LIN {X 0,Y 418.595,Z 415.277,A -85,B 0,C 180,E1 -16911.483,E2 -16911.483} C_VEL
LIN {X 0,Y 414.654,Z 412.078,A -85,B 0,C 180,E1 -16916.405,E2 -16916.405} C_VEL
LIN {X 0,Y 413.753,Z 409.569,A -85,B 0,C 180,E1 -16920.138,E2 -16920.138} C_VEL
LIN {X 0,Y 413.822,Z 409.954,A -85,B 0,C 180,E1 -16922.354,E2 -16922.354} C_VEL
LIN {X 0,Y 418.138,Z 415.092,A -85,B 0,C 180,E1 -16929.775,E2 -16929.775} C_VEL
LIN {X 0,Y 418.882,Z 415.623,A -85,B 0,C 180,E1 -16930.452,E2 -16930.452} C_VEL
LIN {X 0,Y 421.003,Z 419.369,A -85,B 0,C 180,E1 -16932.342,E2 -16932.342} C_VEL
LIN {X 0,Y 424.072,Z 421.923,A -85,B 0,C 180,E1 -16934.404,E2 -16934.404} C_VEL
LIN {X 0,Y 426.834,Z 426.008,A -85,B 0,C 180,E1 -16936.117,E2 -16936.117} C_VEL
LIN {X 0,Y 429.181,Z 428.229,A -85,B 0,C 180,E1 -16937.35,E2 -16937.35} C_VEL
LIN {X 0,Y 432.702,Z 432.705,A -85,B 0,C 180,E1 -16939.086,E2 -16939.086} C_VEL
LIN {X 0,Y 434.181,Z 434.42,A -85,B 0,C 180,E1 -16939.752,E2 -16939.752} C_VEL
LIN {X 0,Y 438.948,Z 440.495,A -85,B 0,C 180,E1 -16941.761,E2 -16941.761} C_VEL
LIN {X 0,Y 444.689,Z 448.712,A -85,B 0,C 180,E1 -16943.945,E2 -16943.945} C_VEL
LIN {X 0,Y 452.263,Z 459.705,A -85,B 0,C 180,E1 -16946.49,E2 -16946.49} C_VEL
LIN {X 0,Y 462.215,Z 475.454,A -85,B 0,C 180,E1 -16949.446,E2 -16949.446} C_VEL
LIN {X 0,Y 471.304,Z 490.869,A -85,B 0,C 180,E1 -16951.853,E2 -16951.853} C_VEL
LIN {X 0,Y 477.792,Z 502.788,A -85,B 0,C 180,E1 -16953.445,E2 -16953.445} C_VEL
LIN {X 0,Y 463.026,Z 751.514,A -85,B 0,C 180,E1 -16957.403,E2 -16957.403} C_VEL
LIN {X 0,Y 460.977,Z 774.068,A -85,B 0,C 180,E1 -16957.838,E2 -16957.838} C_VEL
LIN {X 0,Y 457.627,Z 798.83,A -85,B 0,C 180,E1 -16958.465,E2 -16958.465} C_VEL
LIN {X 0,Y 453.795,Z 820.475,A -85,B 0,C 180,E1 -16959.196,E2 -16959.196} C_VEL
LIN {X 0,Y 449.461,Z 841.373,A -85,B 0,C 180,E1 -16960.068,E2 -16960.068} C_VEL
LIN {X 0,Y 443.769,Z 864.79,A -85,B 0,C 180,E1 -16961.285,E2 -16961.285} C_VEL
LIN {X 0,Y 438.553,Z 883.81,A -85,B 0,C 180,E1 -16962.475,E2 -16962.475} C_VEL
LIN {X 0,Y 431.836,Z 906.004,A -85,B 0,C 180,E1 -16964.128,E2 -16964.128} C_VEL
LIN {X 0,Y 425.724,Z 924.421,A -85,B 0,C 180,E1 -16965.769,E2 -16965.769} C_VEL
LIN {X 0,Y 418.908,Z 943.868,A -85,B 0,C 180,E1 -16967.785,E2 -16967.785} C_VEL
LIN {X 0,Y 412.181,Z 961.726,A -85,B 0,C 180,E1 -16969.995,E2 -16969.995} C_VEL
LIN {X 0,Y 405.9,Z 978.095,A -85,B 0,C 180,E1 -16972.344,E2 -16972.344} C_VEL
LIN {X 0,Y 399.636,Z 994.038,A -85,B 0,C 180,E1 -16975.043,E2 -16975.043} C_VEL
LIN {X 0,Y 394.447,Z 1007.349,A -85,B 0,C 180,E1 -16977.665,E2 -16977.665} C_VEL
LIN {X 0,Y 388.853,Z 1022.095,A -85,B 0,C 180,E1 -16981.091,E2 -16981.091} C_VEL
LIN {X 0,Y 384.923,Z 1033.094,A -85,B 0,C 180,E1 -16984.125,E2 -16984.125} C_VEL
LIN {X 0,Y 381.161,Z 1044.727,A -85,B 0,C 180,E1 -16987.968,E2 -16987.968} C_VEL
LIN {X 0,Y 378.92,Z 1052.817,A -85,B 0,C 180,E1 -16991.22,E2 -16991.22} C_VEL
LIN {X 0,Y 377.195,Z 1060.626,A -85,B 0,C 180,E1 -16995.1,E2 -16995.1} C_VEL
LIN {X 0,Y 376.396,Z 1065.668,A -85,B 0,C 180,E1 -16998.352,E2 -16998.352} C_VEL
LIN {X 0,Y 376.025,Z 1069.646,A -85,B 0,C 180,E1 -17001.744,E2 -17001.744} C_VEL
LIN {X 0,Y 375.948,Z 1072.336,A -85,B 0,C 180,E1 -17005.424,E2 -17005.424} C_VEL
LIN {X 0,Y 375.957,Z 1073.33,A -85,B 0,C 180,E1 -17008.324,E2 -17008.324} C_VEL
LIN {X 0,Y 375.965,Z 1073.331,A -85,B 0,C 180,E1 -17011.219,E2 -17011.219} C_VEL
LIN {X 0,Y 375.951,Z 1072.197,A -85,B 0,C 180,E1 -17014.424,E2 -17014.424} C_VEL
LIN {X 0,Y 376.015,Z 1069.299,A -85,B 0,C 180,E1 -17018.102,E2 -17018.102} C_VEL
LIN {X 0,Y 376.313,Z 1065.625,A -85,B 0,C 180,E1 -17021.184,E2 -17021.184} C_VEL
LIN {X 0,Y 377.065,Z 1060.282,A -85,B 0,C 180,E1 -17024.591,E2 -17024.591} C_VEL
LIN {X 0,Y 378.591,Z 1052.628,A -85,B 0,C 180,E1 -17028.318,E2 -17028.318} C_VEL
LIN {X 0,Y 380.669,Z 1044.446,A -85,B 0,C 180,E1 -17031.576,E2 -17031.576} C_VEL
LIN {X 0,Y 384.037,Z 1033.144,A -85,B 0,C 180,E1 -17035.277,E2 -17035.277} C_VEL
LIN {X 0,Y 387.534,Z 1022.627,A -85,B 0,C 180,E1 -17038.175,E2 -17038.175} C_VEL
LIN {X 0,Y 392.523,Z 1008.535,A -85,B 0,C 180,E1 -17041.48,E2 -17041.48} C_VEL
LIN {X 0,Y 397.395,Z 995.196,A -85,B 0,C 180,E1 -17044.131,E2 -17044.131} C_VEL
LIN {X 0,Y 403.31,Z 979.283,A -85,B 0,C 180,E1 -17046.868,E2 -17046.868} C_VEL
LIN {X 0,Y 409.632,Z 961.81,A -85,B 0,C 180,E1 -17049.394,E2 -17049.394} C_VEL
LIN {X 0,Y 416.292,Z 943.126,A -85,B 0,C 180,E1 -17051.707,E2 -17051.707} C_VEL
LIN {X 0,Y 422.435,Z 924.703,A -85,B 0,C 180,E1 -17053.628,E2 -17053.628} C_VEL
LIN {X 0,Y 428.561,Z 905.351,A -85,B 0,C 180,E1 -17055.366,E2 -17055.366} C_VEL
LIN {X 0,Y 434.811,Z 883.629,A -85,B 0,C 180,E1 -17056.993,E2 -17056.993} C_VEL
LIN {X 0,Y 439.864,Z 864.356,A -85,B 0,C 180,E1 -17058.211,E2 -17058.211} C_VEL
LIN {X 0,Y 445.381,Z 840.47,A -85,B 0,C 180,E1 -17059.459,E2 -17059.459} C_VEL
LIN {X 0,Y 449.404,Z 820.168,A -85,B 0,C 180,E1 -17060.316,E2 -17060.316} C_VEL
LIN {X 0,Y 453.43,Z 796.266,A -85,B 0,C 180,E1 -17061.123,E2 -17061.123} C_VEL
LIN {X 0,Y 456.393,Z 772.598,A -85,B 0,C 180,E1 -17061.714,E2 -17061.714} C_VEL
LIN {X 0,Y 458.46,Z 747.708,A -85,B 0,C 180,E1 -17062.189,E2 -17062.189} C_VEL
LIN {X 0,Y 472.43,Z 499.373,A -85,B 0,C 180,E1 -17066.15,E2 -17066.15} C_VEL
LIN {X 0,Y 462.964,Z 482.094,A -85,B 0,C 180,E1 -17068.344,E2 -17068.344} C_VEL
LIN {X 0,Y 452.861,Z 465.203,A -85,B 0,C 180,E1 -17070.902,E2 -17070.902} C_VEL
LIN {X 0,Y 442.865,Z 449.591,A -85,B 0,C 180,E1 -17073.735,E2 -17073.735} C_VEL
LIN {X 0,Y 433.988,Z 436.811,A -85,B 0,C 180,E1 -17076.582,E2 -17076.582} C_VEL
LIN {X 0,Y 429.245,Z 430.714,A -85,B 0,C 180,E1 -17078.261,E2 -17078.261} C_VEL
LIN {X 0,Y 424.967,Z 425.414,A -85,B 0,C 180,E1 -17079.908,E2 -17079.908} C_VEL
LIN {X 0,Y 421.299,Z 420.825,A -85,B 0,C 180,E1 -17081.456,E2 -17081.456} C_VEL
LIN {X 0,Y 416.853,Z 415.708,A -85,B 0,C 180,E1 -17083.522,E2 -17083.522} C_VEL
LIN {X 0,Y 415.772,Z 414.109,A -85,B 0,C 180,E1 -17084.088,E2 -17084.088} C_VEL
LIN {X 0,Y 412.366,Z 410.911,A -85,B 0,C 180,E1 -17085.908,E2 -17085.908} C_VEL
LIN {X 0,Y 410.586,Z 407.937,A -85,B 0,C 180,E1 -17087.053,E2 -17087.053} C_VEL
LIN {X 0,Y 407.105,Z 405.166,A -85,B 0,C 180,E1 -17089.385,E2 -17089.385} C_VEL
LIN {X 0,Y 405.262,Z 401.53,A -85,B 0,C 180,E1 -17091.058,E2 -17091.058} C_VEL
LIN {X 0,Y 401.47,Z 399.131,A -85,B 0,C 180,E1 -17095.142,E2 -17095.142} C_VEL
LIN {X 0,Y 399.74,Z 395.247,A -85,B 0,C 180,E1 -17100.43,E2 -17100.43} C_VEL
LIN {X 0,Y 399.742,Z 395.247,A -85,B 0,C 180,E1 -17102.007,E2 -17102.007} C_VEL
LIN {X 0,Y 401.877,Z 399.568,A -85,B 0,C 180,E1 -17107.865,E2 -17107.865} C_VEL
LIN {X 0,Y 405.347,Z 401.809,A -85,B 0,C 180,E1 -17111.454,E2 -17111.454} C_VEL
LIN {X 0,Y 407.325,Z 405.383,A -85,B 0,C 180,E1 -17113.197,E2 -17113.197} C_VEL
LIN {X 0,Y 410.405,Z 407.832,A -85,B 0,C 180,E1 -17115.256,E2 -17115.256} C_VEL
LIN {X 0,Y 411.097,Z 408.742,A -85,B 0,C 180,E1 -17115.699,E2 -17115.699} C_VEL
LIN {X 0,Y 413.993,Z 412.767,A -85,B 0,C 180,E1 -17117.427,E2 -17117.427} C_VEL
LIN {X 0,Y 416.281,Z 414.792,A -85,B 0,C 180,E1 -17118.594,E2 -17118.594} C_VEL
LIN {X 0,Y 419.453,Z 418.976,A -85,B 0,C 180,E1 -17120.149,E2 -17120.149} C_VEL
LIN {X 0,Y 421.308,Z 420.811,A -85,B 0,C 180,E1 -17120.964,E2 -17120.964} C_VEL
LIN {X 0,Y 425.07,Z 425.454,A -85,B 0,C 180,E1 -17122.546,E2 -17122.546} C_VEL
LIN {X 0,Y 427.658,Z 428.844,A -85,B 0,C 180,E1 -17123.566,E2 -17123.566} C_VEL
LIN {X 0,Y 431.094,Z 432.964,A -85,B 0,C 180,E1 -17124.823,E2 -17124.823} C_VEL
LIN {X 0,Y 435.975,Z 439.247,A -85,B 0,C 180,E1 -17126.492,E2 -17126.492} C_VEL
LIN {X 0,Y 442.658,Z 447.991,A -85,B 0,C 180,E1 -17128.575,E2 -17128.575} C_VEL
LIN {X 0,Y 452.49,Z 461.584,A -85,B 0,C 180,E1 -17131.322,E2 -17131.322} C_VEL
LIN {X 0,Y 462.744,Z 476.797,A -85,B 0,C 180,E1 -17133.882,E2 -17133.882} C_VEL
LIN {X 0,Y 472.66,Z 492.479,A -85,B 0,C 180,E1 -17136.128,E2 -17136.128} C_VEL
LIN {X 0,Y 458.588,Z 739.184,A -85,B 0,C 180,E1 -17140.069,E2 -17140.069} C_VEL
LIN {X 0,Y 456.64,Z 761.14,A -85,B 0,C 180,E1 -17140.516,E2 -17140.516} C_VEL
LIN {X 0,Y 453.326,Z 786.702,A -85,B 0,C 180,E1 -17141.231,E2 -17141.231} C_VEL
LIN {X 0,Y 450.006,Z 806.703,A -85,B 0,C 180,E1 -17141.956,E2 -17141.956} C_VEL
LIN {X 0,Y 445.549,Z 829.565,A -85,B 0,C 180,E1 -17142.979,E2 -17142.979} C_VEL
LIN {X 0,Y 440.536,Z 851.049,A -85,B 0,C 180,E1 -17144.174,E2 -17144.174} C_VEL
LIN {X 0,Y 435.215,Z 871.436,A -85,B 0,C 180,E1 -17145.515,E2 -17145.515} C_VEL
LIN {X 0,Y 428.993,Z 892.708,A -85,B 0,C 180,E1 -17147.201,E2 -17147.201} C_VEL
LIN {X 0,Y 423.304,Z 910.614,A -85,B 0,C 180,E1 -17148.864,E2 -17148.864} C_VEL
LIN {X 0,Y 416.422,Z 930.803,A -85,B 0,C 180,E1 -17151.076,E2 -17151.076} C_VEL
LIN {X 0,Y 410.742,Z 946.551,A -85,B 0,C 180,E1 -17153.099,E2 -17153.099} C_VEL
LIN {X 0,Y 404.223,Z 964.023,A -85,B 0,C 180,E1 -17155.709,E2 -17155.709} C_VEL
LIN {X 0,Y 398.77,Z 978.285,A -85,B 0,C 180,E1 -17158.227,E2 -17158.227} C_VEL
LIN {X 0,Y 393.418,Z 992.492,A -85,B 0,C 180,E1 -17161.126,E2 -17161.126} C_VEL
LIN {X 0,Y 388.636,Z 1005.189,A -85,B 0,C 180,E1 -17164.227,E2 -17164.227} C_VEL
LIN {X 0,Y 384.759,Z 1016.241,A -85,B 0,C 180,E1 -17167.38,E2 -17167.38} C_VEL
LIN {X 0,Y 381.461,Z 1026.344,A -85,B 0,C 180,E1 -17170.874,E2 -17170.874} C_VEL
LIN {X 0,Y 379.252,Z 1034.079,A -85,B 0,C 180,E1 -17174.086,E2 -17174.086} C_VEL
LIN {X 0,Y 377.506,Z 1041.462,A -85,B 0,C 180,E1 -17177.922,E2 -17177.922} C_VEL
LIN {X 0,Y 376.635,Z 1046.231,A -85,B 0,C 180,E1 -17181.142,E2 -17181.142} C_VEL
LIN {X 0,Y 376.175,Z 1050.124,A -85,B 0,C 180,E1 -17184.662,E2 -17184.662} C_VEL
LIN {X 0,Y 376.006,Z 1052.412,A -85,B 0,C 180,E1 -17188.171,E2 -17188.171} C_VEL
LIN {X 0,Y 375.97,Z 1053.298,A -85,B 0,C 180,E1 -17191.067,E2 -17191.067} C_VEL
LIN {X 0,Y 375.98,Z 1053.205,A -85,B 0,C 180,E1 -17194.219,E2 -17194.219} C_VEL
LIN {X 0,Y 376.077,Z 1051.718,A -85,B 0,C 180,E1 -17197.793,E2 -17197.793} C_VEL
LIN {X 0,Y 376.362,Z 1049.06,A -85,B 0,C 180,E1 -17201.028,E2 -17201.028} C_VEL
LIN {X 0,Y 376.991,Z 1045.229,A -85,B 0,C 180,E1 -17204.28,E2 -17204.28} C_VEL
LIN {X 0,Y 378.403,Z 1038.971,A -85,B 0,C 180,E1 -17208.168,E2 -17208.168} C_VEL
LIN {X 0,Y 380.312,Z 1032.182,A -85,B 0,C 180,E1 -17211.453,E2 -17211.453} C_VEL
LIN {X 0,Y 383.447,Z 1022.659,A -85,B 0,C 180,E1 -17215.196,E2 -17215.196} C_VEL
LIN {X 0,Y 384.449,Z 1019.742,A -85,B 0,C 180,E1 -17216.188,E2 -17216.188} C_VEL
LIN {X 0,Y 384.646,Z 1016.77,A -85,B 0,C 180,E1 -17217.254,E2 -17217.254} C_VEL
LIN {X 0,Y 382.131,Z 1008.67,A -85,B 0,C 180,E1 -17220.166,E2 -17220.166} C_VEL
LIN {X 0,Y 382.694,Z 1005.603,A -85,B 0,C 180,E1 -17221.052,E2 -17221.052} C_VEL
LIN {X 0,Y 388.256,Z 992.368,A -85,B 0,C 180,E1 -17224.333,E2 -17224.333} C_VEL
LIN {X 0,Y 394.017,Z 978.627,A -85,B 0,C 180,E1 -17227.171,E2 -17227.171} C_VEL
LIN {X 0,Y 400.549,Z 963.213,A -85,B 0,C 180,E1 -17229.907,E2 -17229.907} C_VEL
LIN {X 0,Y 407.452,Z 946.166,A -85,B 0,C 180,E1 -17232.443,E2 -17232.443} C_VEL
LIN {X 0,Y 414.186,Z 929.038,A -85,B 0,C 180,E1 -17234.628,E2 -17234.628} C_VEL
LIN {X 0,Y 421.151,Z 910.027,A -85,B 0,C 180,E1 -17236.674,E2 -17236.674} C_VEL
LIN {X 0,Y 427.212,Z 892.368,A -85,B 0,C 180,E1 -17238.298,E2 -17238.298} C_VEL
LIN {X 0,Y 434.282,Z 869.687,A -85,B 0,C 180,E1 -17240.058,E2 -17240.058} C_VEL
LIN {X 0,Y 439.772,Z 850.01,A -85,B 0,C 180,E1 -17241.325,E2 -17241.325} C_VEL
LIN {X 0,Y 445.565,Z 826.246,A -85,B 0,C 180,E1 -17242.6,E2 -17242.6} C_VEL
LIN {X 0,Y 449.848,Z 805.433,A -85,B 0,C 180,E1 -17243.498,E2 -17243.498} C_VEL
LIN {X 0,Y 453.959,Z 781.735,A -85,B 0,C 180,E1 -17244.321,E2 -17244.321} C_VEL
LIN {X 0,Y 457.039,Z 757.598,A -85,B 0,C 180,E1 -17244.941,E2 -17244.941} C_VEL
LIN {X 0,Y 459.217,Z 732.893,A -85,B 0,C 180,E1 -17245.412,E2 -17245.412} C_VEL
LIN {X 0,Y 473.455,Z 500.104,A -85,B 0,C 180,E1 -17249.123,E2 -17249.123} C_VEL
LIN {X 0,Y 463.328,Z 484.174,A -85,B 0,C 180,E1 -17251.697,E2 -17251.697} C_VEL
LIN {X 0,Y 453.867,Z 470.442,A -85,B 0,C 180,E1 -17254.383,E2 -17254.383} C_VEL
LIN {X 0,Y 446.179,Z 459.921,A -85,B 0,C 180,E1 -17256.84,E2 -17256.84} C_VEL
LIN {X 0,Y 439.936,Z 451.462,A -85,B 0,C 180,E1 -17259.094,E2 -17259.094} C_VEL
LIN {X 0,Y 435.12,Z 445.449,A -85,B 0,C 180,E1 -17261.025,E2 -17261.025} C_VEL
LIN {X 0,Y 431.297,Z 440.548,A -85,B 0,C 180,E1 -17262.738,E2 -17262.738} C_VEL
LIN {X 0,Y 427.805,Z 436.18,A -85,B 0,C 180,E1 -17264.477,E2 -17264.477} C_VEL
LIN {X 0,Y 426.589,Z 434.763,A -85,B 0,C 180,E1 -17265.128,E2 -17265.128} C_VEL
LIN {X 0,Y 423.245,Z 430.774,A -85,B 0,C 180,E1 -17267.1,E2 -17267.1} C_VEL
LIN {X 0,Y 422.373,Z 429.307,A -85,B 0,C 180,E1 -17267.698,E2 -17267.698} C_VEL
LIN {X 0,Y 418.943,Z 426.044,A -85,B 0,C 180,E1 -17270.174,E2 -17270.174} C_VEL
LIN {X 0,Y 417.474,Z 423.172,A -85,B 0,C 180,E1 -17271.599,E2 -17271.599} C_VEL
LIN {X 0,Y 413.613,Z 419.955,A -85,B 0,C 180,E1 -17276.535,E2 -17276.535} C_VEL
LIN {X 0,Y 412.773,Z 417.456,A -85,B 0,C 180,E1 -17280.278,E2 -17280.278} C_VEL
LIN {X 0,Y 412.842,Z 417.936,A -85,B 0,C 180,E1 -17282.36,E2 -17282.36} C_VEL
LIN {X 0,Y 417.027,Z 422.988,A -85,B 0,C 180,E1 -17289.662,E2 -17289.662} C_VEL
LIN {X 0,Y 417.682,Z 423.496,A -85,B 0,C 180,E1 -17290.273,E2 -17290.273} C_VEL
LIN {X 0,Y 419.856,Z 427.269,A -85,B 0,C 180,E1 -17292.237,E2 -17292.237} C_VEL
LIN {X 0,Y 422.682,Z 429.677,A -85,B 0,C 180,E1 -17294.172,E2 -17294.172} C_VEL
LIN {X 0,Y 425.518,Z 433.819,A -85,B 0,C 180,E1 -17295.958,E2 -17295.958} C_VEL
LIN {X 0,Y 427.645,Z 435.902,A -85,B 0,C 180,E1 -17297.099,E2 -17297.099} C_VEL
LIN {X 0,Y 431.324,Z 440.528,A -85,B 0,C 180,E1 -17298.938,E2 -17298.938} C_VEL
LIN {X 0,Y 437.04,Z 447.87,A -85,B 0,C 180,E1 -17301.438,E2 -17301.438} C_VEL
LIN {X 0,Y 442.601,Z 455.989,A -85,B 0,C 180,E1 -17303.605,E2 -17303.605} C_VEL
LIN {X 0,Y 449.951,Z 466.899,A -85,B 0,C 180,E1 -17306.136,E2 -17306.136} C_VEL
LIN {X 0,Y 459.467,Z 482.19,A -85,B 0,C 180,E1 -17309.032,E2 -17309.032} C_VEL
LIN {X 0,Y 468.305,Z 497.46,A -85,B 0,C 180,E1 -17311.433,E2 -17311.433} C_VEL
LIN {X 0,Y 473.26,Z 506.669,A -85,B 0,C 180,E1 -17312.69,E2 -17312.69} C_VEL
LIN {X 0,Y 458.137,Z 753.356,A -85,B 0,C 180,E1 -17316.632,E2 -17316.632} C_VEL
LIN {X 0,Y 455.983,Z 775.737,A -85,B 0,C 180,E1 -17317.072,E2 -17317.072} C_VEL
LIN {X 0,Y 452.153,Z 802.073,A -85,B 0,C 180,E1 -17317.764,E2 -17317.764} C_VEL
LIN {X 0,Y 448.34,Z 822.781,A -85,B 0,C 180,E1 -17318.482,E2 -17318.482} C_VEL
LIN {X 0,Y 443.19,Z 846.317,A -85,B 0,C 180,E1 -17319.503,E2 -17319.503} C_VEL
LIN {X 0,Y 437.935,Z 866.84,A -85,B 0,C 180,E1 -17320.61,E2 -17320.61} C_VEL
LIN {X 0,Y 432.081,Z 887.426,A -85,B 0,C 180,E1 -17321.928,E2 -17321.928} C_VEL
LIN {X 0,Y 425.546,Z 907.928,A -85,B 0,C 180,E1 -17323.508,E2 -17323.508} C_VEL
LIN {X 0,Y 419.209,Z 926.381,A -85,B 0,C 180,E1 -17325.185,E2 -17325.185} C_VEL
LIN {X 0,Y 411.637,Z 946.918,A -85,B 0,C 180,E1 -17327.393,E2 -17327.393} C_VEL
LIN {X 0,Y 405.349,Z 963.072,A -85,B 0,C 180,E1 -17329.443,E2 -17329.443} C_VEL
LIN {X 0,Y 398.317,Z 980.667,A -85,B 0,C 180,E1 -17332.047,E2 -17332.047} C_VEL
LIN {X 0,Y 392.19,Z 995.609,A -85,B 0,C 180,E1 -17334.671,E2 -17334.671} C_VEL
LIN {X 0,Y 386.377,Z 1010.038,A -85,B 0,C 180,E1 -17337.609,E2 -17337.609} C_VEL
LIN {X 0,Y 381.166,Z 1023.104,A -85,B 0,C 180,E1 -17340.796,E2 -17340.796} C_VEL
LIN {X 0,Y 376.92,Z 1034.573,A -85,B 0,C 180,E1 -17344.066,E2 -17344.066} C_VEL
LIN {X 0,Y 373.388,Z 1044.968,A -85,B 0,C 180,E1 -17347.65,E2 -17347.65} C_VEL
LIN {X 0,Y 371.048,Z 1053,A -85,B 0,C 180,E1 -17350.97,E2 -17350.97} C_VEL
LIN {X 0,Y 369.244,Z 1060.698,A -85,B 0,C 180,E1 -17354.932,E2 -17354.932} C_VEL
LIN {X 0,Y 368.41,Z 1065.687,A -85,B 0,C 180,E1 -17358.255,E2 -17358.255} C_VEL
LIN {X 0,Y 368.013,Z 1069.776,A -85,B 0,C 180,E1 -17361.878,E2 -17361.878} C_VEL
LIN {X 0,Y 367.949,Z 1072.2,A -85,B 0,C 180,E1 -17365.48,E2 -17365.48} C_VEL
LIN {X 0,Y 367.96,Z 1073.142,A -85,B 0,C 180,E1 -17368.443,E2 -17368.443} C_VEL
LIN {X 0,Y 367.964,Z 1073.092,A -85,B 0,C 180,E1 -17371.401,E2 -17371.401} C_VEL
LIN {X 0,Y 367.957,Z 1071.742,A -85,B 0,C 180,E1 -17374.989,E2 -17374.989} C_VEL
LIN {X 0,Y 368.049,Z 1068.787,A -85,B 0,C 180,E1 -17378.546,E2 -17378.546} C_VEL
LIN {X 0,Y 368.399,Z 1064.96,A -85,B 0,C 180,E1 -17381.745,E2 -17381.745} C_VEL
LIN {X 0,Y 369.37,Z 1058.884,A -85,B 0,C 180,E1 -17385.545,E2 -17385.545} C_VEL
LIN {X 0,Y 370.963,Z 1051.643,A -85,B 0,C 180,E1 -17389.035,E2 -17389.035} C_VEL
LIN {X 0,Y 373.52,Z 1042.506,A -85,B 0,C 180,E1 -17392.673,E2 -17392.673} C_VEL
LIN {X 0,Y 376.915,Z 1031.81,A -85,B 0,C 180,E1 -17396.127,E2 -17396.127} C_VEL
LIN {X 0,Y 381.193,Z 1019.77,A -85,B 0,C 180,E1 -17399.441,E2 -17399.441} C_VEL
LIN {X 0,Y 386.259,Z 1006.087,A -85,B 0,C 180,E1 -17402.577,E2 -17402.577} C_VEL
LIN {X 0,Y 391.772,Z 991.744,A -85,B 0,C 180,E1 -17405.405,E2 -17405.405} C_VEL
LIN {X 0,Y 398.151,Z 975.046,A -85,B 0,C 180,E1 -17408.182,E2 -17408.182} C_VEL
LIN {X 0,Y 404.06,Z 959.404,A -85,B 0,C 180,E1 -17410.417,E2 -17410.417} C_VEL
LIN {X 0,Y 411.225,Z 939.668,A -85,B 0,C 180,E1 -17412.812,E2 -17412.812} C_VEL
LIN {X 0,Y 417.284,Z 922.041,A -85,B 0,C 180,E1 -17414.629,E2 -17414.629} C_VEL
LIN {X 0,Y 424.273,Z 900.17,A -85,B 0,C 180,E1 -17416.541,E2 -17416.541} C_VEL
LIN {X 0,Y 429.916,Z 880.895,A -85,B 0,C 180,E1 -17417.946,E2 -17417.946} C_VEL
LIN {X 0,Y 435.801,Z 858.702,A -85,B 0,C 180,E1 -17419.314,E2 -17419.314} C_VEL
LIN {X 0,Y 440.76,Z 836.985,A -85,B 0,C 180,E1 -17420.397,E2 -17420.397} C_VEL
LIN {X 0,Y 444.916,Z 816.254,A -85,B 0,C 180,E1 -17421.245,E2 -17421.245} C_VEL
LIN {X 0,Y 449.001,Z 791.127,A -85,B 0,C 180,E1 -17422.045,E2 -17422.045} C_VEL
LIN {X 0,Y 451.686,Z 769.398,A -85,B 0,C 180,E1 -17422.569,E2 -17422.569} C_VEL
LIN {X 0,Y 454.074,Z 736.841,A -85,B 0,C 180,E1 -17423.153,E2 -17423.153} C_VEL
LIN {X 0,Y 467.644,Z 503.033,A -85,B 0,C 180,E1 -17426.899,E2 -17426.899} C_VEL
LIN {X 0,Y 457.829,Z 485.159,A -85,B 0,C 180,E1 -17429.266,E2 -17429.266} C_VEL
LIN {X 0,Y 448.434,Z 469.378,A -85,B 0,C 180,E1 -17431.754,E2 -17431.754} C_VEL
LIN {X 0,Y 439.686,Z 455.676,A -85,B 0,C 180,E1 -17434.328,E2 -17434.328} C_VEL
LIN {X 0,Y 431.475,Z 443.557,A -85,B 0,C 180,E1 -17437.052,E2 -17437.052} C_VEL
LIN {X 0,Y 427.074,Z 437.891,A -85,B 0,C 180,E1 -17438.65,E2 -17438.65} C_VEL
LIN {X 0,Y 423.034,Z 432.801,A -85,B 0,C 180,E1 -17440.245,E2 -17440.245} C_VEL
LIN {X 0,Y 419.299,Z 427.956,A -85,B 0,C 180,E1 -17441.868,E2 -17441.868} C_VEL
LIN {X 0,Y 415.399,Z 423.561,A -85,B 0,C 180,E1 -17443.715,E2 -17443.715} C_VEL
LIN {X 0,Y 414.009,Z 421.639,A -85,B 0,C 180,E1 -17444.45,E2 -17444.45} C_VEL
LIN {X 0,Y 410.724,Z 418.316,A -85,B 0,C 180,E1 -17446.269,E2 -17446.269} C_VEL
LIN {X 0,Y 409.172,Z 415.703,A -85,B 0,C 180,E1 -17447.295,E2 -17447.295} C_VEL
LIN {X 0,Y 405.686,Z 412.733,A -85,B 0,C 180,E1 -17449.707,E2 -17449.707} C_VEL
LIN {X 0,Y 403.962,Z 409.372,A -85,B 0,C 180,E1 -17451.316,E2 -17451.316} C_VEL
LIN {X 0,Y 400.228,Z 406.777,A -85,B 0,C 180,E1 -17455.558,E2 -17455.558} C_VEL
LIN {X 0,Y 398.765,Z 403.19,A -85,B 0,C 180,E1 -17460.431,E2 -17460.431} C_VEL
LIN {X 0,Y 398.764,Z 403.218,A -85,B 0,C 180,E1 -17462.012,E2 -17462.012} C_VEL
LIN {X 0,Y 402.905,Z 408.947,A -85,B 0,C 180,E1 -17470.149,E2 -17470.149} C_VEL
LIN {X 0,Y 404.064,Z 409.552,A -85,B 0,C 180,E1 -17471.201,E2 -17471.201} C_VEL
LIN {X 0,Y 406.171,Z 413.304,A -85,B 0,C 180,E1 -17473.09,E2 -17473.09} C_VEL
LIN {X 0,Y 409.485,Z 416.11,A -85,B 0,C 180,E1 -17475.327,E2 -17475.327} C_VEL
LIN {X 0,Y 412.414,Z 420.34,A -85,B 0,C 180,E1 -17477.132,E2 -17477.132} C_VEL
LIN {X 0,Y 414.717,Z 422.496,A -85,B 0,C 180,E1 -17478.339,E2 -17478.339} C_VEL
LIN {X 0,Y 418.065,Z 426.807,A -85,B 0,C 180,E1 -17480,E2 -17480} C_VEL
LIN {X 0,Y 419.667,Z 428.537,A -85,B 0,C 180,E1 -17480.721,E2 -17480.721} C_VEL
LIN {X 0,Y 423.636,Z 433.301,A -85,B 0,C 180,E1 -17482.407,E2 -17482.407} C_VEL
LIN {X 0,Y 429.418,Z 440.849,A -85,B 0,C 180,E1 -17484.633,E2 -17484.633} C_VEL
LIN {X 0,Y 434.165,Z 447.01,A -85,B 0,C 180,E1 -17486.28,E2 -17486.28} C_VEL
LIN {X 0,Y 440.974,Z 456.175,A -85,B 0,C 180,E1 -17488.436,E2 -17488.436} C_VEL
LIN {X 0,Y 449.772,Z 468.497,A -85,B 0,C 180,E1 -17490.937,E2 -17490.937} C_VEL
LIN {X 0,Y 459.776,Z 483.553,A -85,B 0,C 180,E1 -17493.493,E2 -17493.493} C_VEL
LIN {X 0,Y 467.865,Z 496.717,A -85,B 0,C 180,E1 -17495.389,E2 -17495.389} C_VEL
LIN {X 0,Y 453.549,Z 740.077,A -85,B 0,C 180,E1 -17499.294,E2 -17499.294} C_VEL
LIN {X 0,Y 451.468,Z 762.645,A -85,B 0,C 180,E1 -17499.76,E2 -17499.76} C_VEL
LIN {X 0,Y 448.099,Z 787.565,A -85,B 0,C 180,E1 -17500.469,E2 -17500.469} C_VEL
LIN {X 0,Y 444.73,Z 807.283,A -85,B 0,C 180,E1 -17501.188,E2 -17501.188} C_VEL
LIN {X 0,Y 439.958,Z 830.893,A -85,B 0,C 180,E1 -17502.258,E2 -17502.258} C_VEL
LIN {X 0,Y 434.991,Z 851.578,A -85,B 0,C 180,E1 -17503.417,E2 -17503.417} C_VEL
LIN {X 0,Y 429.294,Z 872.789,A -85,B 0,C 180,E1 -17504.824,E2 -17504.824} C_VEL
LIN {X 0,Y 423.117,Z 893.156,A -85,B 0,C 180,E1 -17506.46,E2 -17506.46} C_VEL
LIN {X 0,Y 417.04,Z 911.701,A -85,B 0,C 180,E1 -17508.2,E2 -17508.2} C_VEL
LIN {X 0,Y 410.018,Z 931.561,A -85,B 0,C 180,E1 -17510.409,E2 -17510.409} C_VEL
LIN {X 0,Y 404.138,Z 947.318,A -85,B 0,C 180,E1 -17512.462,E2 -17512.462} C_VEL
LIN {X 0,Y 397.273,Z 965.01,A -85,B 0,C 180,E1 -17515.157,E2 -17515.157} C_VEL
LIN {X 0,Y 391.57,Z 979.385,A -85,B 0,C 180,E1 -17517.745,E2 -17517.745} C_VEL
LIN {X 0,Y 385.699,Z 994.267,A -85,B 0,C 180,E1 -17520.885,E2 -17520.885} C_VEL
LIN {X 0,Y 381.095,Z 1006.064,A -85,B 0,C 180,E1 -17523.846,E2 -17523.846} C_VEL
LIN {X 0,Y 376.909,Z 1017.523,A -85,B 0,C 180,E1 -17527.212,E2 -17527.212} C_VEL
LIN {X 0,Y 373.528,Z 1027.42,A -85,B 0,C 180,E1 -17530.776,E2 -17530.776} C_VEL
LIN {X 0,Y 371.105,Z 1035.73,A -85,B 0,C 180,E1 -17534.369,E2 -17534.369} C_VEL
LIN {X 0,Y 369.496,Z 1042.216,A -85,B 0,C 180,E1 -17537.973,E2 -17537.973} C_VEL
LIN {X 0,Y 368.621,Z 1046.883,A -85,B 0,C 180,E1 -17541.263,E2 -17541.263} C_VEL
LIN {X 0,Y 368.137,Z 1050.811,A -85,B 0,C 180,E1 -17545.17,E2 -17545.17} C_VEL
LIN {X 0,Y 368.003,Z 1052.77,A -85,B 0,C 180,E1 -17548.443,E2 -17548.443} C_VEL
LIN {X 0,Y 367.963,Z 1053.583,A -85,B 0,C 180,E1 -17551.557,E2 -17551.557} C_VEL
LIN {X 0,Y 367.998,Z 1053.234,A -85,B 0,C 180,E1 -17555.144,E2 -17555.144} C_VEL
LIN {X 0,Y 368.14,Z 1051.47,A -85,B 0,C 180,E1 -17558.591,E2 -17558.591} C_VEL
LIN {X 0,Y 368.47,Z 1048.781,A -85,B 0,C 180,E1 -17561.743,E2 -17561.743} C_VEL
LIN {X 0,Y 369.381,Z 1044.115,A -85,B 0,C 180,E1 -17565.545,E2 -17565.545} C_VEL
LIN {X 0,Y 370.849,Z 1038.244,A -85,B 0,C 180,E1 -17569.041,E2 -17569.041} C_VEL
LIN {X 0,Y 373.227,Z 1030.64,A -85,B 0,C 180,E1 -17572.692,E2 -17572.692} C_VEL
LIN {X 0,Y 376.569,Z 1021.105,A -85,B 0,C 180,E1 -17576.323,E2 -17576.323} C_VEL
LIN {X 0,Y 380.596,Z 1010.851,A -85,B 0,C 180,E1 -17579.598,E2 -17579.598} C_VEL
LIN {X 0,Y 382.694,Z 1005.603,A -85,B 0,C 180,E1 -17581.052,E2 -17581.052} C_VEL
LIN {X 0,Y 383.317,Z 1002.103,A -85,B 0,C 180,E1 -17582.081,E2 -17582.081} C_VEL
LIN {X 0,Y 381.972,Z 992.669,A -85,B 0,C 180,E1 -17584.925,E2 -17584.925} C_VEL
LIN {X 0,Y 382.854,Z 989.136,A -85,B 0,C 180,E1 -17585.766,E2 -17585.766} C_VEL
LIN {X 0,Y 388.792,Z 975.723,A -85,B 0,C 180,E1 -17588.49,E2 -17588.49} C_VEL
LIN {X 0,Y 395.749,Z 959.633,A -85,B 0,C 180,E1 -17591.257,E2 -17591.257} C_VEL
LIN {X 0,Y 402.235,Z 944.199,A -85,B 0,C 180,E1 -17593.518,E2 -17593.518} C_VEL
LIN {X 0,Y 409.965,Z 924.952,A -85,B 0,C 180,E1 -17595.912,E2 -17595.912} C_VEL
LIN {X 0,Y 416.614,Z 907.166,A -85,B 0,C 180,E1 -17597.777,E2 -17597.777} C_VEL
LIN {X 0,Y 423.872,Z 886.302,A -85,B 0,C 180,E1 -17599.635,E2 -17599.635} C_VEL
LIN {X 0,Y 429.927,Z 866.82,A -85,B 0,C 180,E1 -17601.084,E2 -17601.084} C_VEL
LIN {X 0,Y 436.219,Z 844.593,A -85,B 0,C 180,E1 -17602.475,E2 -17602.475} C_VEL
LIN {X 0,Y 441.487,Z 822.45,A -85,B 0,C 180,E1 -17603.602,E2 -17603.602} C_VEL
LIN {X 0,Y 445.876,Z 801.155,A -85,B 0,C 180,E1 -17604.492,E2 -17604.492} C_VEL
LIN {X 0,Y 449.985,Z 776.229,A -85,B 0,C 180,E1 -17605.301,E2 -17605.301} C_VEL
LIN {X 0,Y 452.78,Z 754.059,A -85,B 0,C 180,E1 -17605.843,E2 -17605.843} C_VEL
LIN {X 0,Y 455.317,Z 721.258,A -85,B 0,C 180,E1 -17606.422,E2 -17606.422} C_VEL
LIN {X 0,Y 469.023,Z 504.436,A -85,B 0,C 180,E1 -17609.881,E2 -17609.881} C_VEL
LIN {X 0,Y 459.73,Z 489.717,A -85,B 0,C 180,E1 -17612.332,E2 -17612.332} C_VEL
LIN {X 0,Y 451.14,Z 477.063,A -85,B 0,C 180,E1 -17614.85,E2 -17614.85} C_VEL
LIN {X 0,Y 443.696,Z 466.703,A -85,B 0,C 180,E1 -17617.299,E2 -17617.299} C_VEL
LIN {X 0,Y 437.661,Z 458.472,A -85,B 0,C 180,E1 -17619.54,E2 -17619.54} C_VEL
LIN {X 0,Y 433.252,Z 452.826,A -85,B 0,C 180,E1 -17621.359,E2 -17621.359} C_VEL
LIN {X 0,Y 429.5,Z 447.972,A -85,B 0,C 180,E1 -17623.082,E2 -17623.082} C_VEL
LIN {X 0,Y 425.925,Z 443.233,A -85,B 0,C 180,E1 -17624.93,E2 -17624.93} C_VEL
LIN {X 0,Y 421.947,Z 438.647,A -85,B 0,C 180,E1 -17627.268,E2 -17627.268} C_VEL
LIN {X 0,Y 420.99,Z 437.062,A -85,B 0,C 180,E1 -17627.936,E2 -17627.936} C_VEL
LIN {X 0,Y 417.57,Z 433.613,A -85,B 0,C 180,E1 -17630.49,E2 -17630.49} C_VEL
LIN {X 0,Y 416.205,Z 431.007,A -85,B 0,C 180,E1 -17631.851,E2 -17631.851} C_VEL
LIN {X 0,Y 412.17,Z 427.007,A -85,B 0,C 180,E1 -17637.775,E2 -17637.775} C_VEL
LIN {X 0,Y 411.795,Z 425.299,A -85,B 0,C 180,E1 -17640.556,E2 -17640.556} C_VEL
LIN {X 0,Y 411.898,Z 426.108,A -85,B 0,C 180,E1 -17642.644,E2 -17642.644} C_VEL
LIN {X 0,Y 415.919,Z 430.884,A -85,B 0,C 180,E1 -17649.548,E2 -17649.548} C_VEL
LIN {X 0,Y 416.55,Z 431.513,A -85,B 0,C 180,E1 -17650.162,E2 -17650.162} C_VEL
LIN {X 0,Y 418.885,Z 435.355,A -85,B 0,C 180,E1 -17652.266,E2 -17652.266} C_VEL
LIN {X 0,Y 421.301,Z 437.421,A -85,B 0,C 180,E1 -17653.939,E2 -17653.939} C_VEL
LIN {X 0,Y 424.321,Z 441.746,A -85,B 0,C 180,E1 -17655.864,E2 -17655.864} C_VEL
LIN {X 0,Y 426.118,Z 443.564,A -85,B 0,C 180,E1 -17656.846,E2 -17656.846} C_VEL
LIN {X 0,Y 429.95,Z 448.349,A -85,B 0,C 180,E1 -17658.79,E2 -17658.79} C_VEL
LIN {X 0,Y 435.295,Z 455.466,A -85,B 0,C 180,E1 -17661.175,E2 -17661.175} C_VEL
LIN {X 0,Y 440.693,Z 463.515,A -85,B 0,C 180,E1 -17663.324,E2 -17663.324} C_VEL
LIN {X 0,Y 447.764,Z 474.27,A -85,B 0,C 180,E1 -17665.814,E2 -17665.814} C_VEL
LIN {X 0,Y 456.781,Z 488.986,A -85,B 0,C 180,E1 -17668.624,E2 -17668.624} C_VEL
LIN {X 0,Y 465.329,Z 504.068,A -85,B 0,C 180,E1 -17671.009,E2 -17671.009} C_VEL
LIN {X 0,Y 468.796,Z 510.797,A -85,B 0,C 180,E1 -17671.923,E2 -17671.923} C_VEL
LIN {X 0,Y 453.357,Z 754.88,A -85,B 0,C 180,E1 -17675.839,E2 -17675.839} C_VEL
LIN {X 0,Y 450.926,Z 778.675,A -85,B 0,C 180,E1 -17676.316,E2 -17676.316} C_VEL
LIN {X 0,Y 447.1,Z 803.382,A -85,B 0,C 180,E1 -17676.986,E2 -17676.986} C_VEL
LIN {X 0,Y 443.092,Z 824.425,A -85,B 0,C 180,E1 -17677.726,E2 -17677.726} C_VEL
LIN {X 0,Y 437.526,Z 848.652,A -85,B 0,C 180,E1 -17678.804,E2 -17678.804} C_VEL
LIN {X 0,Y 432.44,Z 867.888,A -85,B 0,C 180,E1 -17679.857,E2 -17679.857} C_VEL
LIN {X 0,Y 425.904,Z 890.012,A -85,B 0,C 180,E1 -17681.3,E2 -17681.3} C_VEL
LIN {X 0,Y 419.385,Z 909.625,A -85,B 0,C 180,E1 -17682.85,E2 -17682.85} C_VEL
LIN {X 0,Y 412.739,Z 928.342,A -85,B 0,C 180,E1 -17684.583,E2 -17684.583} C_VEL
LIN {X 0,Y 405.103,Z 948.175,A -85,B 0,C 180,E1 -17686.769,E2 -17686.769} C_VEL
LIN {X 0,Y 398.482,Z 964.6,A -85,B 0,C 180,E1 -17688.896,E2 -17688.896} C_VEL
LIN {X 0,Y 391.099,Z 982.254,A -85,B 0,C 180,E1 -17691.592,E2 -17691.592} C_VEL
LIN {X 0,Y 385.189,Z 996.151,A -85,B 0,C 180,E1 -17694.087,E2 -17694.087} C_VEL
LIN {X 0,Y 378.842,Z 1011.201,A -85,B 0,C 180,E1 -17697.244,E2 -17697.244} C_VEL
LIN {X 0,Y 373.719,Z 1023.535,A -85,B 0,C 180,E1 -17700.332,E2 -17700.332} C_VEL
LIN {X 0,Y 369.151,Z 1035.366,A -85,B 0,C 180,E1 -17703.8,E2 -17703.8} C_VEL
LIN {X 0,Y 365.626,Z 1045.209,A -85,B 0,C 180,E1 -17707.319,E2 -17707.319} C_VEL
LIN {X 0,Y 363.088,Z 1053.541,A -85,B 0,C 180,E1 -17710.87,E2 -17710.87} C_VEL
LIN {X 0,Y 361.296,Z 1060.77,A -85,B 0,C 180,E1 -17714.757,E2 -17714.757} C_VEL
LIN {X 0,Y 360.425,Z 1065.706,A -85,B 0,C 180,E1 -17718.153,E2 -17718.153} C_VEL
LIN {X 0,Y 360.004,Z 1069.826,A -85,B 0,C 180,E1 -17722.017,E2 -17722.017} C_VEL
LIN {X 0,Y 359.952,Z 1071.994,A -85,B 0,C 180,E1 -17725.379,E2 -17725.379} C_VEL
LIN {X 0,Y 359.962,Z 1072.932,A -85,B 0,C 180,E1 -17728.408,E2 -17728.408} C_VEL
LIN {X 0,Y 359.966,Z 1072.875,A -85,B 0,C 180,E1 -17731.432,E2 -17731.432} C_VEL
LIN {X 0,Y 359.958,Z 1071.612,A -85,B 0,C 180,E1 -17734.94,E2 -17734.94} C_VEL
LIN {X 0,Y 360.053,Z 1068.647,A -85,B 0,C 180,E1 -17738.644,E2 -17738.644} C_VEL
LIN {X 0,Y 360.413,Z 1064.93,A -85,B 0,C 180,E1 -17741.847,E2 -17741.847} C_VEL
LIN {X 0,Y 361.408,Z 1059.041,A -85,B 0,C 180,E1 -17745.677,E2 -17745.677} C_VEL
LIN {X 0,Y 363.091,Z 1051.74,A -85,B 0,C 180,E1 -17749.297,E2 -17749.297} C_VEL
LIN {X 0,Y 365.622,Z 1043.077,A -85,B 0,C 180,E1 -17752.851,E2 -17752.851} C_VEL
LIN {X 0,Y 369.3,Z 1032.048,A -85,B 0,C 180,E1 -17756.535,E2 -17756.535} C_VEL
LIN {X 0,Y 373.422,Z 1020.87,A -85,B 0,C 180,E1 -17759.694,E2 -17759.694} C_VEL
LIN {X 0,Y 379.003,Z 1006.487,A -85,B 0,C 180,E1 -17763.1,E2 -17763.1} C_VEL
LIN {X 0,Y 384.385,Z 992.988,A -85,B 0,C 180,E1 -17765.823,E2 -17765.823} C_VEL
LIN {X 0,Y 391.357,Z 975.51,A -85,B 0,C 180,E1 -17768.807,E2 -17768.807} C_VEL
LIN {X 0,Y 397.396,Z 960.08,A -85,B 0,C 180,E1 -17771.049,E2 -17771.049} C_VEL
LIN {X 0,Y 404.992,Z 939.906,A -85,B 0,C 180,E1 -17773.537,E2 -17773.537} C_VEL
LIN {X 0,Y 411.158,Z 922.544,A -85,B 0,C 180,E1 -17775.346,E2 -17775.346} C_VEL
LIN {X 0,Y 418.181,Z 901.381,A -85,B 0,C 180,E1 -17777.227,E2 -17777.227} C_VEL
LIN {X 0,Y 424.222,Z 881.357,A -85,B 0,C 180,E1 -17778.703,E2 -17778.703} C_VEL
LIN {X 0,Y 430.263,Z 859.322,A -85,B 0,C 180,E1 -17780.075,E2 -17780.075} C_VEL
LIN {X 0,Y 435.549,Z 836.78,A -85,B 0,C 180,E1 -17781.205,E2 -17781.205} C_VEL
LIN {X 0,Y 439.892,Z 815.654,A -85,B 0,C 180,E1 -17782.068,E2 -17782.068} C_VEL
LIN {X 0,Y 444.032,Z 790.684,A -85,B 0,C 180,E1 -17782.859,E2 -17782.859} C_VEL
LIN {X 0,Y 446.787,Z 768.832,A -85,B 0,C 180,E1 -17783.384,E2 -17783.384} C_VEL
LIN {X 0,Y 449.223,Z 736.198,A -85,B 0,C 180,E1 -17783.969,E2 -17783.969} C_VEL
LIN {X 0,Y 462.934,Z 506.831,A -85,B 0,C 180,E1 -17787.661,E2 -17787.661} C_VEL
LIN {X 0,Y 453.675,Z 489.843,A -85,B 0,C 180,E1 -17789.98,E2 -17789.98} C_VEL
LIN {X 0,Y 445.019,Z 475.093,A -85,B 0,C 180,E1 -17792.356,E2 -17792.356} C_VEL
LIN {X 0,Y 436.749,Z 462.007,A -85,B 0,C 180,E1 -17794.869,E2 -17794.869} C_VEL
LIN {X 0,Y 429.076,Z 450.432,A -85,B 0,C 180,E1 -17797.495,E2 -17797.495} C_VEL
LIN {X 0,Y 424.757,Z 444.874,A -85,B 0,C 180,E1 -17799.106,E2 -17799.106} C_VEL
LIN {X 0,Y 421.117,Z 440.183,A -85,B 0,C 180,E1 -17800.585,E2 -17800.585} C_VEL
LIN {X 0,Y 416.87,Z 434.813,A -85,B 0,C 180,E1 -17802.481,E2 -17802.481} C_VEL
LIN {X 0,Y 413.273,Z 430.311,A -85,B 0,C 180,E1 -17804.277,E2 -17804.277} C_VEL
LIN {X 0,Y 412.265,Z 429.153,A -85,B 0,C 180,E1 -17804.815,E2 -17804.815} C_VEL
LIN {X 0,Y 408.976,Z 425.523,A -85,B 0,C 180,E1 -17806.714,E2 -17806.714} C_VEL
LIN {X 0,Y 407.766,Z 423.461,A -85,B 0,C 180,E1 -17807.538,E2 -17807.538} C_VEL
LIN {X 0,Y 404.364,Z 420.418,A -85,B 0,C 180,E1 -17809.96,E2 -17809.96} C_VEL
LIN {X 0,Y 402.672,Z 417.207,A -85,B 0,C 180,E1 -17811.576,E2 -17811.576} C_VEL
LIN {X 0,Y 399.086,Z 414.532,A -85,B 0,C 180,E1 -17815.833,E2 -17815.833} C_VEL
LIN {X 0,Y 397.781,Z 411.103,A -85,B 0,C 180,E1 -17820.576,E2 -17820.576} C_VEL
LIN {X 0,Y 397.785,Z 411.188,A -85,B 0,C 180,E1 -17822.017,E2 -17822.017} C_VEL
LIN {X 0,Y 401.797,Z 416.836,A -85,B 0,C 180,E1 -17830.032,E2 -17830.032} C_VEL
LIN {X 0,Y 402.918,Z 417.633,A -85,B 0,C 180,E1 -17831.089,E2 -17831.089} C_VEL
LIN {X 0,Y 405.199,Z 421.43,A -85,B 0,C 180,E1 -17833.122,E2 -17833.122} C_VEL
LIN {X 0,Y 408.13,Z 423.971,A -85,B 0,C 180,E1 -17835.125,E2 -17835.125} C_VEL
LIN {X 0,Y 411.209,Z 428.274,A -85,B 0,C 180,E1 -17837.038,E2 -17837.038} C_VEL
LIN {X 0,Y 413.164,Z 430.186,A -85,B 0,C 180,E1 -17838.082,E2 -17838.082} C_VEL
LIN {X 0,Y 416.681,Z 434.634,A -85,B 0,C 180,E1 -17839.85,E2 -17839.85} C_VEL
LIN {X 0,Y 418.245,Z 436.571,A -85,B 0,C 180,E1 -17840.575,E2 -17840.575} C_VEL
LIN {X 0,Y 422.722,Z 442.153,A -85,B 0,C 180,E1 -17842.495,E2 -17842.495} C_VEL
LIN {X 0,Y 427.325,Z 448.118,A -85,B 0,C 180,E1 -17844.283,E2 -17844.283} C_VEL
LIN {X 0,Y 433.757,Z 456.516,A -85,B 0,C 180,E1 -17846.528,E2 -17846.528} C_VEL
LIN {X 0,Y 443.951,Z 470.767,A -85,B 0,C 180,E1 -17849.665,E2 -17849.665} C_VEL
LIN {X 0,Y 453.574,Z 485.262,A -85,B 0,C 180,E1 -17852.279,E2 -17852.279} C_VEL
LIN {X 0,Y 463.165,Z 500.599,A -85,B 0,C 180,E1 -17854.627,E2 -17854.627} C_VEL
LIN {X 0,Y 448.659,Z 740.144,A -85,B 0,C 180,E1 -17858.489,E2 -17858.489} C_VEL
LIN {X 0,Y 446.546,Z 762.536,A -85,B 0,C 180,E1 -17858.951,E2 -17858.951} C_VEL
LIN {X 0,Y 443.089,Z 787.592,A -85,B 0,C 180,E1 -17859.661,E2 -17859.661} C_VEL
LIN {X 0,Y 439.523,Z 807.94,A -85,B 0,C 180,E1 -17860.405,E2 -17860.405} C_VEL
LIN {X 0,Y 434.441,Z 832.213,A -85,B 0,C 180,E1 -17861.518,E2 -17861.518} C_VEL
LIN {X 0,Y 429.506,Z 852.174,A -85,B 0,C 180,E1 -17862.645,E2 -17862.645} C_VEL
LIN {X 0,Y 423.414,Z 874.165,A -85,B 0,C 180,E1 -17864.119,E2 -17864.119} C_VEL
LIN {X 0,Y 417.077,Z 894.328,A -85,B 0,C 180,E1 -17865.762,E2 -17865.762} C_VEL
LIN {X 0,Y 410.614,Z 913.446,A -85,B 0,C 180,E1 -17867.583,E2 -17867.583} C_VEL
LIN {X 0,Y 403.671,Z 932.318,A -85,B 0,C 180,E1 -17869.722,E2 -17869.722} C_VEL
LIN {X 0,Y 397.633,Z 947.961,A -85,B 0,C 180,E1 -17871.787,E2 -17871.787} C_VEL
LIN {X 0,Y 390.277,Z 966.194,A -85,B 0,C 180,E1 -17874.619,E2 -17874.619} C_VEL
LIN {X 0,Y 384.706,Z 979.727,A -85,B 0,C 180,E1 -17877.097,E2 -17877.097} C_VEL
LIN {X 0,Y 378.679,Z 994.392,A -85,B 0,C 180,E1 -17880.237,E2 -17880.237} C_VEL
LIN {X 0,Y 373.754,Z 1006.473,A -85,B 0,C 180,E1 -17883.322,E2 -17883.322} C_VEL
LIN {X 0,Y 369.412,Z 1017.815,A -85,B 0,C 180,E1 -17886.723,E2 -17886.723} C_VEL
LIN {X 0,Y 365.987,Z 1027.307,A -85,B 0,C 180,E1 -17890.198,E2 -17890.198} C_VEL
LIN {X 0,Y 363.389,Z 1035.666,A -85,B 0,C 180,E1 -17893.865,E2 -17893.865} C_VEL
LIN {X 0,Y 361.597,Z 1042.474,A -85,B 0,C 180,E1 -17897.706,E2 -17897.706} C_VEL
LIN {X 0,Y 360.667,Z 1047.132,A -85,B 0,C 180,E1 -17901.069,E2 -17901.069} C_VEL
LIN {X 0,Y 360.15,Z 1051.044,A -85,B 0,C 180,E1 -17905.063,E2 -17905.063} C_VEL
LIN {X 0,Y 360.011,Z 1052.928,A -85,B 0,C 180,E1 -17908.249,E2 -17908.249} C_VEL
LIN {X 0,Y 359.971,Z 1053.755,A -85,B 0,C 180,E1 -17911.273,E2 -17911.273} C_VEL
LIN {X 0,Y 359.993,Z 1053.576,A -85,B 0,C 180,E1 -17914.78,E2 -17914.78} C_VEL
LIN {X 0,Y 360.142,Z 1051.888,A -85,B 0,C 180,E1 -17918.462,E2 -17918.462} C_VEL
LIN {X 0,Y 360.474,Z 1049.252,A -85,B 0,C 180,E1 -17921.716,E2 -17921.716} C_VEL
LIN {X 0,Y 361.347,Z 1044.99,A -85,B 0,C 180,E1 -17925.405,E2 -17925.405} C_VEL
LIN {X 0,Y 362.996,Z 1038.712,A -85,B 0,C 180,E1 -17929.302,E2 -17929.302} C_VEL
LIN {X 0,Y 365.225,Z 1031.847,A -85,B 0,C 180,E1 -17932.707,E2 -17932.707} C_VEL
LIN {X 0,Y 368.807,Z 1022.158,A -85,B 0,C 180,E1 -17936.573,E2 -17936.573} C_VEL
LIN {X 0,Y 372.735,Z 1012.517,A -85,B 0,C 180,E1 -17939.754,E2 -17939.754} C_VEL
LIN {X 0,Y 378.376,Z 999.354,A -85,B 0,C 180,E1 -17943.378,E2 -17943.378} C_VEL
LIN {X 0,Y 382.854,Z 989.136,A -85,B 0,C 180,E1 -17945.766,E2 -17945.766} C_VEL
LIN {X 0,Y 383.853,Z 985.086,A -85,B 0,C 180,E1 -17946.74,E2 -17946.74} C_VEL
LIN {X 0,Y 383.625,Z 974.33,A -85,B 0,C 180,E1 -17949.478,E2 -17949.478} C_VEL
LIN {X 0,Y 384.786,Z 970.371,A -85,B 0,C 180,E1 -17950.26,E2 -17950.26} C_VEL
LIN {X 0,Y 391.207,Z 956.01,A -85,B 0,C 180,E1 -17952.634,E2 -17952.634} C_VEL
LIN {X 0,Y 398.981,Z 937.989,A -85,B 0,C 180,E1 -17955.172,E2 -17955.172} C_VEL
LIN {X 0,Y 405.645,Z 921.531,A -85,B 0,C 180,E1 -17957.131,E2 -17957.131} C_VEL
LIN {X 0,Y 412.922,Z 902.567,A -85,B 0,C 180,E1 -17959.07,E2 -17959.07} C_VEL
LIN {X 0,Y 419.945,Z 882.198,A -85,B 0,C 180,E1 -17960.807,E2 -17960.807} C_VEL
LIN {X 0,Y 425.953,Z 863.235,A -85,B 0,C 180,E1 -17962.177,E2 -17962.177} C_VEL
LIN {X 0,Y 432.451,Z 839.933,A -85,B 0,C 180,E1 -17963.574,E2 -17963.574} C_VEL
LIN {X 0,Y 437.087,Z 820.715,A -85,B 0,C 180,E1 -17964.527,E2 -17964.527} C_VEL
LIN {X 0,Y 441.996,Z 796.971,A -85,B 0,C 180,E1 -17965.488,E2 -17965.488} C_VEL
LIN {X 0,Y 445.667,Z 774.241,A -85,B 0,C 180,E1 -17966.197,E2 -17966.197} C_VEL
LIN {X 0,Y 448.734,Z 749.707,A -85,B 0,C 180,E1 -17966.775,E2 -17966.775} C_VEL
LIN {X 0,Y 452.235,Z 698.908,A -85,B 0,C 180,E1 -17967.622,E2 -17967.622} C_VEL
LIN {X 0,Y 464.59,Z 508.604,A -85,B 0,C 180,E1 -17970.677,E2 -17970.677} C_VEL
LIN {X 0,Y 455.479,Z 494.085,A -85,B 0,C 180,E1 -17973.184,E2 -17973.184} C_VEL
LIN {X 0,Y 446.434,Z 480.677,A -85,B 0,C 180,E1 -17975.979,E2 -17975.979} C_VEL
LIN {X 0,Y 438.584,Z 469.793,A -85,B 0,C 180,E1 -17978.747,E2 -17978.747} C_VEL
LIN {X 0,Y 434.792,Z 464.712,A -85,B 0,C 180,E1 -17980.241,E2 -17980.241} C_VEL
LIN {X 0,Y 431.544,Z 460.364,A -85,B 0,C 180,E1 -17981.632,E2 -17981.632} C_VEL
LIN {X 0,Y 427.72,Z 455.387,A -85,B 0,C 180,E1 -17983.429,E2 -17983.429} C_VEL
LIN {X 0,Y 423.811,Z 450.255,A -85,B 0,C 180,E1 -17985.517,E2 -17985.517} C_VEL
LIN {X 0,Y 420.368,Z 446.019,A -85,B 0,C 180,E1 -17987.639,E2 -17987.639} C_VEL
LIN {X 0,Y 419.414,Z 444.673,A -85,B 0,C 180,E1 -17988.308,E2 -17988.308} C_VEL
LIN {X 0,Y 416.067,Z 440.931,A -85,B 0,C 180,E1 -17990.943,E2 -17990.943} C_VEL
LIN {X 0,Y 414.944,Z 438.835,A -85,B 0,C 180,E1 -17992.105,E2 -17992.105} C_VEL
LIN {X 0,Y 410.991,Z 434.346,A -85,B 0,C 180,E1 -17998.606,E2 -17998.606} C_VEL
LIN {X 0,Y 410.809,Z 433.294,A -85,B 0,C 180,E1 -18000.837,E2 -18000.837} C_VEL
LIN {X 0,Y 410.994,Z 434.348,A -85,B 0,C 180,E1 -18003.068,E2 -18003.068} C_VEL
LIN {X 0,Y 414.811,Z 438.779,A -85,B 0,C 180,E1 -18009.434,E2 -18009.434} C_VEL
LIN {X 0,Y 415.358,Z 439.369,A -85,B 0,C 180,E1 -18009.981,E2 -18009.981} C_VEL
LIN {X 0,Y 417.74,Z 443.249,A -85,B 0,C 180,E1 -18012.16,E2 -18012.16} C_VEL
LIN {X 0,Y 420.018,Z 445.339,A -85,B 0,C 180,E1 -18013.772,E2 -18013.772} C_VEL
LIN {X 0,Y 423.126,Z 449.666,A -85,B 0,C 180,E1 -18015.769,E2 -18015.769} C_VEL
LIN {X 0,Y 424.657,Z 451.317,A -85,B 0,C 180,E1 -18016.624,E2 -18016.624} C_VEL
LIN {X 0,Y 429.284,Z 457.356,A -85,B 0,C 180,E1 -18018.993,E2 -18018.993} C_VEL
LIN {X 0,Y 433.486,Z 462.944,A -85,B 0,C 180,E1 -18020.878,E2 -18020.878} C_VEL
LIN {X 0,Y 438.796,Z 471.036,A -85,B 0,C 180,E1 -18023.04,E2 -18023.04} C_VEL
LIN {X 0,Y 445.496,Z 481.462,A -85,B 0,C 180,E1 -18025.456,E2 -18025.456} C_VEL
LIN {X 0,Y 454.24,Z 495.979,A -85,B 0,C 180,E1 -18028.247,E2 -18028.247} C_VEL
LIN {X 0,Y 462.483,Z 510.87,A -85,B 0,C 180,E1 -18030.608,E2 -18030.608} C_VEL
LIN {X 0,Y 464.434,Z 514.678,A -85,B 0,C 180,E1 -18031.139,E2 -18031.139} C_VEL
LIN {X 0,Y 448.744,Z 755.445,A -85,B 0,C 180,E1 -18035.012,E2 -18035.012} C_VEL
LIN {X 0,Y 446.107,Z 780.197,A -85,B 0,C 180,E1 -18035.513,E2 -18035.513} C_VEL
LIN {X 0,Y 442.178,Z 804.436,A -85,B 0,C 180,E1 -18036.183,E2 -18036.183} C_VEL
LIN {X 0,Y 437.618,Z 827.548,A -85,B 0,C 180,E1 -18037.008,E2 -18037.008} C_VEL
LIN {X 0,Y 431.928,Z 850.988,A -85,B 0,C 180,E1 -18038.086,E2 -18038.086} C_VEL
LIN {X 0,Y 426.407,Z 871.122,A -85,B 0,C 180,E1 -18039.214,E2 -18039.214} C_VEL
LIN {X 0,Y 419.487,Z 893.253,A -85,B 0,C 180,E1 -18040.713,E2 -18040.713} C_VEL
LIN {X 0,Y 413.371,Z 911.069,A -85,B 0,C 180,E1 -18042.151,E2 -18042.151} C_VEL
LIN {X 0,Y 405.816,Z 931.508,A -85,B 0,C 180,E1 -18044.092,E2 -18044.092} C_VEL
LIN {X 0,Y 398.479,Z 949.77,A -85,B 0,C 180,E1 -18046.167,E2 -18046.167} C_VEL
LIN {X 0,Y 391.064,Z 967.555,A -85,B 0,C 180,E1 -18048.53,E2 -18048.53} C_VEL
LIN {X 0,Y 383.78,Z 984.132,A -85,B 0,C 180,E1 -18051.17,E2 -18051.17} C_VEL
LIN {X 0,Y 377.203,Z 999.1,A -85,B 0,C 180,E1 -18053.951,E2 -18053.951} C_VEL
LIN {X 0,Y 370.747,Z 1013.623,A -85,B 0,C 180,E1 -18057.174,E2 -18057.174} C_VEL
LIN {X 0,Y 365.59,Z 1025.702,A -85,B 0,C 180,E1 -18060.328,E2 -18060.328} C_VEL
LIN {X 0,Y 360.788,Z 1037.528,A -85,B 0,C 180,E1 -18064.031,E2 -18064.031} C_VEL
LIN {X 0,Y 357.556,Z 1046.378,A -85,B 0,C 180,E1 -18067.344,E2 -18067.344} C_VEL
LIN {X 0,Y 354.658,Z 1055.63,A -85,B 0,C 180,E1 -18071.593,E2 -18071.593} C_VEL
LIN {X 0,Y 353.183,Z 1061.621,A -85,B 0,C 180,E1 -18075.071,E2 -18075.071} C_VEL
LIN {X 0,Y 352.279,Z 1066.928,A -85,B 0,C 180,E1 -18079.037,E2 -18079.037} C_VEL
LIN {X 0,Y 351.995,Z 1070.211,A -85,B 0,C 180,E1 -18082.656,E2 -18082.656} C_VEL
LIN {X 0,Y 351.951,Z 1071.999,A -85,B 0,C 180,E1 -18085.764,E2 -18085.764} C_VEL
LIN {X 0,Y 351.973,Z 1072.815,A -85,B 0,C 180,E1 -18089.023,E2 -18089.023} C_VEL
LIN {X 0,Y 351.967,Z 1072.366,A -85,B 0,C 180,E1 -18092.768,E2 -18092.768} C_VEL
LIN {X 0,Y 351.967,Z 1070.589,A -85,B 0,C 180,E1 -18096.197,E2 -18096.197} C_VEL
LIN {X 0,Y 352.107,Z 1067.776,A -85,B 0,C 180,E1 -18099.48,E2 -18099.48} C_VEL
LIN {X 0,Y 352.731,Z 1062.919,A -85,B 0,C 180,E1 -18103.441,E2 -18103.441} C_VEL
LIN {X 0,Y 353.947,Z 1056.822,A -85,B 0,C 180,E1 -18107.085,E2 -18107.085} C_VEL
LIN {X 0,Y 355.965,Z 1049.31,A -85,B 0,C 180,E1 -18110.728,E2 -18110.728} C_VEL
LIN {X 0,Y 359.067,Z 1039.611,A -85,B 0,C 180,E1 -18114.514,E2 -18114.514} C_VEL
LIN {X 0,Y 362.686,Z 1029.662,A -85,B 0,C 180,E1 -18117.769,E2 -18117.769} C_VEL
LIN {X 0,Y 367.966,Z 1016.219,A -85,B 0,C 180,E1 -18121.448,E2 -18121.448} C_VEL
LIN {X 0,Y 373.183,Z 1003.477,A -85,B 0,C 180,E1 -18124.387,E2 -18124.387} C_VEL
LIN {X 0,Y 380.209,Z 986.613,A -85,B 0,C 180,E1 -18127.666,E2 -18127.666} C_VEL
LIN {X 0,Y 386.364,Z 971.686,A -85,B 0,C 180,E1 -18130.121,E2 -18130.121} C_VEL
LIN {X 0,Y 393.942,Z 952.789,A -85,B 0,C 180,E1 -18132.762,E2 -18132.762} C_VEL
LIN {X 0,Y 400.418,Z 935.829,A -85,B 0,C 180,E1 -18134.764,E2 -18134.764} C_VEL
LIN {X 0,Y 407.616,Z 916.009,A -85,B 0,C 180,E1 -18136.765,E2 -18136.765} C_VEL
LIN {X 0,Y 414.205,Z 896.031,A -85,B 0,C 180,E1 -18138.447,E2 -18138.447} C_VEL
LIN {X 0,Y 420.649,Z 875,A -85,B 0,C 180,E1 -18139.942,E2 -18139.942} C_VEL
LIN {X 0,Y 426.695,Z 852.212,A -85,B 0,C 180,E1 -18141.268,E2 -18141.268} C_VEL
LIN {X 0,Y 431.897,Z 830.068,A -85,B 0,C 180,E1 -18142.324,E2 -18142.324} C_VEL
LIN {X 0,Y 436.586,Z 805.872,A -85,B 0,C 180,E1 -18143.227,E2 -18143.227} C_VEL
LIN {X 0,Y 440.126,Z 783.489,A -85,B 0,C 180,E1 -18143.872,E2 -18143.872} C_VEL
LIN {X 0,Y 442.965,Z 757.691,A -85,B 0,C 180,E1 -18144.425,E2 -18144.425} C_VEL
LIN {X 0,Y 457.195,Z 528.6,A -85,B 0,C 180,E1 -18148.145,E2 -18148.145} C_VEL
LIN {X 0,Y 458.241,Z 510.448,A -85,B 0,C 180,E1 -18148.457,E2 -18148.457} C_VEL
LIN {X 0,Y 449.907,Z 495.126,A -85,B 0,C 180,E1 -18150.62,E2 -18150.62} C_VEL
LIN {X 0,Y 442.152,Z 481.656,A -85,B 0,C 180,E1 -18152.819,E2 -18152.819} C_VEL
LIN {X 0,Y 434.226,Z 468.876,A -85,B 0,C 180,E1 -18155.295,E2 -18155.295} C_VEL
LIN {X 0,Y 426.87,Z 457.577,A -85,B 0,C 180,E1 -18157.881,E2 -18157.881} C_VEL
LIN {X 0,Y 422.631,Z 452.038,A -85,B 0,C 180,E1 -18159.503,E2 -18159.503} C_VEL
LIN {X 0,Y 419.215,Z 447.562,A -85,B 0,C 180,E1 -18160.927,E2 -18160.927} C_VEL
LIN {X 0,Y 415.047,Z 442.231,A -85,B 0,C 180,E1 -18162.836,E2 -18162.836} C_VEL
LIN {X 0,Y 411.423,Z 437.457,A -85,B 0,C 180,E1 -18164.711,E2 -18164.711} C_VEL
LIN {X 0,Y 407.56,Z 433.226,A -85,B 0,C 180,E1 -18166.955,E2 -18166.955} C_VEL
LIN {X 0,Y 406.369,Z 431.211,A -85,B 0,C 180,E1 -18167.783,E2 -18167.783} C_VEL
LIN {X 0,Y 403.049,Z 428.102,A -85,B 0,C 180,E1 -18170.216,E2 -18170.216} C_VEL
LIN {X 0,Y 401.547,Z 425.1,A -85,B 0,C 180,E1 -18171.696,E2 -18171.696} C_VEL
LIN {X 0,Y 397.954,Z 422.286,A -85,B 0,C 180,E1 -18176.11,E2 -18176.11} C_VEL
LIN {X 0,Y 396.799,Z 419.017,A -85,B 0,C 180,E1 -18180.722,E2 -18180.722} C_VEL
LIN {X 0,Y 396.807,Z 419.157,A -85,B 0,C 180,E1 -18182.022,E2 -18182.022} C_VEL
LIN {X 0,Y 400.691,Z 424.725,A -85,B 0,C 180,E1 -18189.915,E2 -18189.915} C_VEL
LIN {X 0,Y 401.649,Z 425.352,A -85,B 0,C 180,E1 -18190.834,E2 -18190.834} C_VEL
LIN {X 0,Y 404.048,Z 429.334,A -85,B 0,C 180,E1 -18193.015,E2 -18193.015} C_VEL
LIN {X 0,Y 406.735,Z 431.719,A -85,B 0,C 180,E1 -18194.886,E2 -18194.886} C_VEL
LIN {X 0,Y 409.885,Z 436.086,A -85,B 0,C 180,E1 -18196.876,E2 -18196.876} C_VEL
LIN {X 0,Y 411.619,Z 437.865,A -85,B 0,C 180,E1 -18197.823,E2 -18197.823} C_VEL
LIN {X 0,Y 415.157,Z 442.327,A -85,B 0,C 180,E1 -18199.632,E2 -18199.632} C_VEL
LIN {X 0,Y 420.881,Z 449.647,A -85,B 0,C 180,E1 -18202.194,E2 -18202.194} C_VEL
LIN {X 0,Y 425.498,Z 455.738,A -85,B 0,C 180,E1 -18204.025,E2 -18204.025} C_VEL
LIN {X 0,Y 431.574,Z 463.827,A -85,B 0,C 180,E1 -18206.191,E2 -18206.191} C_VEL
LIN {X 0,Y 441.424,Z 477.827,A -85,B 0,C 180,E1 -18209.293,E2 -18209.293} C_VEL
LIN {X 0,Y 450.695,Z 492.011,A -85,B 0,C 180,E1 -18211.872,E2 -18211.872} C_VEL
LIN {X 0,Y 458.538,Z 504.882,A -85,B 0,C 180,E1 -18213.86,E2 -18213.86} C_VEL
LIN {X 0,Y 443.713,Z 742.048,A -85,B 0,C 180,E1 -18217.698,E2 -18217.698} C_VEL
LIN {X 0,Y 441.261,Z 766.52,A -85,B 0,C 180,E1 -18218.219,E2 -18218.219} C_VEL
LIN {X 0,Y 437.81,Z 789.774,A -85,B 0,C 180,E1 -18218.907,E2 -18218.907} C_VEL
LIN {X 0,Y 433.999,Z 810.733,A -85,B 0,C 180,E1 -18219.691,E2 -18219.691} C_VEL
LIN {X 0,Y 428.732,Z 834.62,A -85,B 0,C 180,E1 -18220.817,E2 -18220.817} C_VEL
LIN {X 0,Y 423.61,Z 854.622,A -85,B 0,C 180,E1 -18221.967,E2 -18221.967} C_VEL
LIN {X 0,Y 416.833,Z 877.841,A -85,B 0,C 180,E1 -18223.579,E2 -18223.579} C_VEL
LIN {X 0,Y 410.859,Z 896.225,A -85,B 0,C 180,E1 -18225.109,E2 -18225.109} C_VEL
LIN {X 0,Y 403.772,Z 916.375,A -85,B 0,C 180,E1 -18227.078,E2 -18227.078} C_VEL
LIN {X 0,Y 397.097,Z 933.804,A -85,B 0,C 180,E1 -18229.105,E2 -18229.105} C_VEL
LIN {X 0,Y 390.107,Z 951.336,A -85,B 0,C 180,E1 -18231.476,E2 -18231.476} C_VEL
LIN {X 0,Y 382.956,Z 968.211,A -85,B 0,C 180,E1 -18234.207,E2 -18234.207} C_VEL
LIN {X 0,Y 376.637,Z 983.099,A -85,B 0,C 180,E1 -18237.028,E2 -18237.028} C_VEL
LIN {X 0,Y 370.529,Z 997.207,A -85,B 0,C 180,E1 -18240.229,E2 -18240.229} C_VEL
LIN {X 0,Y 365.459,Z 1009.343,A -85,B 0,C 180,E1 -18243.466,E2 -18243.466} C_VEL
LIN {X 0,Y 361.02,Z 1020.354,A -85,B 0,C 180,E1 -18247.013,E2 -18247.013} C_VEL
LIN {X 0,Y 357.798,Z 1029.176,A -85,B 0,C 180,E1 -18250.406,E2 -18250.406} C_VEL
LIN {X 0,Y 355.037,Z 1037.749,A -85,B 0,C 180,E1 -18254.482,E2 -18254.482} C_VEL
LIN {X 0,Y 353.529,Z 1043.476,A -85,B 0,C 180,E1 -18257.919,E2 -18257.919} C_VEL
LIN {X 0,Y 352.54,Z 1048.508,A -85,B 0,C 180,E1 -18261.847,E2 -18261.847} C_VEL
LIN {X 0,Y 352.13,Z 1051.608,A -85,B 0,C 180,E1 -18265.44,E2 -18265.44} C_VEL
LIN {X 0,Y 352.007,Z 1053.352,A -85,B 0,C 180,E1 -18268.698,E2 -18268.698} C_VEL
LIN {X 0,Y 351.971,Z 1054.11,A -85,B 0,C 180,E1 -18272.279,E2 -18272.279} C_VEL
LIN {X 0,Y 352.032,Z 1053.375,A -85,B 0,C 180,E1 -18276.033,E2 -18276.033} C_VEL
LIN {X 0,Y 352.203,Z 1051.642,A -85,B 0,C 180,E1 -18279.313,E2 -18279.313} C_VEL
LIN {X 0,Y 352.745,Z 1048.383,A -85,B 0,C 180,E1 -18283.107,E2 -18283.107} C_VEL
LIN {X 0,Y 353.89,Z 1043.468,A -85,B 0,C 180,E1 -18286.919,E2 -18286.919} C_VEL
LIN {X 0,Y 355.635,Z 1037.688,A -85,B 0,C 180,E1 -18290.404,E2 -18290.404} C_VEL
LIN {X 0,Y 358.748,Z 1028.987,A -85,B 0,C 180,E1 -18294.537,E2 -18294.537} C_VEL
LIN {X 0,Y 362.176,Z 1020.487,A -85,B 0,C 180,E1 -18297.812,E2 -18297.812} C_VEL
LIN {X 0,Y 367.254,Z 1008.837,A -85,B 0,C 180,E1 -18301.55,E2 -18301.55} C_VEL
LIN {X 0,Y 372.564,Z 997.067,A -85,B 0,C 180,E1 -18304.678,E2 -18304.678} C_VEL
LIN {X 0,Y 378.856,Z 983.488,A -85,B 0,C 180,E1 -18307.756,E2 -18307.756} C_VEL
LIN {X 0,Y 384.786,Z 970.371,A -85,B 0,C 180,E1 -18310.26,E2 -18310.26} C_VEL
LIN {X 0,Y 386.11,Z 965.772,A -85,B 0,C 180,E1 -18311.166,E2 -18311.166} C_VEL
LIN {X 0,Y 386.856,Z 953.733,A -85,B 0,C 180,E1 -18313.759,E2 -18313.759} C_VEL
LIN {X 0,Y 388.217,Z 949.36,A -85,B 0,C 180,E1 -18314.474,E2 -18314.474} C_VEL
LIN {X 0,Y 395.316,Z 933.042,A -85,B 0,C 180,E1 -18316.651,E2 -18316.651} C_VEL
LIN {X 0,Y 403.19,Z 913.925,A -85,B 0,C 180,E1 -18318.822,E2 -18318.822} C_VEL
LIN {X 0,Y 410.223,Z 895.262,A -85,B 0,C 180,E1 -18320.594,E2 -18320.594} C_VEL
LIN {X 0,Y 417.332,Z 874.846,A -85,B 0,C 180,E1 -18322.246,E2 -18322.246} C_VEL
LIN {X 0,Y 423.901,Z 853.376,A -85,B 0,C 180,E1 -18323.672,E2 -18323.672} C_VEL
LIN {X 0,Y 429.437,Z 832.992,A -85,B 0,C 180,E1 -18324.811,E2 -18324.811} C_VEL
LIN {X 0,Y 435.035,Z 808.649,A -85,B 0,C 180,E1 -18325.908,E2 -18325.908} C_VEL
LIN {X 0,Y 439.077,Z 787.492,A -85,B 0,C 180,E1 -18326.664,E2 -18326.664} C_VEL
LIN {X 0,Y 442.89,Z 761.686,A -85,B 0,C 180,E1 -18327.37,E2 -18327.37} C_VEL
LIN {X 0,Y 445.135,Z 739.577,A -85,B 0,C 180,E1 -18327.813,E2 -18327.813} C_VEL
LIN {X 0,Y 460.357,Z 513.032,A -85,B 0,C 180,E1 -18331.456,E2 -18331.456} C_VEL
LIN {X 0,Y 452.087,Z 499.823,A -85,B 0,C 180,E1 -18333.817,E2 -18333.817} C_VEL
LIN {X 0,Y 444.077,Z 487.694,A -85,B 0,C 180,E1 -18336.372,E2 -18336.372} C_VEL
LIN {X 0,Y 436.457,Z 476.937,A -85,B 0,C 180,E1 -18339.13,E2 -18339.13} C_VEL
LIN {X 0,Y 432.367,Z 471.377,A -85,B 0,C 180,E1 -18340.794,E2 -18340.794} C_VEL
LIN {X 0,Y 429.562,Z 467.569,A -85,B 0,C 180,E1 -18342.036,E2 -18342.036} C_VEL
LIN {X 0,Y 426.088,Z 462.935,A -85,B 0,C 180,E1 -18343.714,E2 -18343.714} C_VEL
LIN {X 0,Y 422.253,Z 457.842,A -85,B 0,C 180,E1 -18345.813,E2 -18345.813} C_VEL
LIN {X 0,Y 418.806,Z 453.389,A -85,B 0,C 180,E1 -18348.012,E2 -18348.012} C_VEL
LIN {X 0,Y 417.858,Z 452.262,A -85,B 0,C 180,E1 -18348.684,E2 -18348.684} C_VEL
LIN {X 0,Y 414.659,Z 448.361,A -85,B 0,C 180,E1 -18351.332,E2 -18351.332} C_VEL
LIN {X 0,Y 413.833,Z 446.725,A -85,B 0,C 180,E1 -18352.224,E2 -18352.224} C_VEL
LIN {X 0,Y 409.966,Z 442.107,A -85,B 0,C 180,E1 -18358.882,E2 -18358.882} C_VEL
LIN {X 0,Y 409.832,Z 441.261,A -85,B 0,C 180,E1 -18360.979,E2 -18360.979} C_VEL
LIN {X 0,Y 410.141,Z 442.736,A -85,B 0,C 180,E1 -18363.634,E2 -18363.634} C_VEL
LIN {X 0,Y 413.848,Z 446.734,A -85,B 0,C 180,E1 -18369.456,E2 -18369.456} C_VEL
LIN {X 0,Y 416.772,Z 451.317,A -85,B 0,C 180,E1 -18372.188,E2 -18372.188} C_VEL
LIN {X 0,Y 418.651,Z 453.067,A -85,B 0,C 180,E1 -18373.536,E2 -18373.536} C_VEL
LIN {X 0,Y 421.818,Z 457.472,A -85,B 0,C 180,E1 -18375.607,E2 -18375.607} C_VEL
LIN {X 0,Y 423.204,Z 459.062,A -85,B 0,C 180,E1 -18376.4,E2 -18376.4} C_VEL
LIN {X 0,Y 427.636,Z 464.936,A -85,B 0,C 180,E1 -18378.718,E2 -18378.718} C_VEL
LIN {X 0,Y 431.762,Z 470.528,A -85,B 0,C 180,E1 -18380.61,E2 -18380.61} C_VEL
LIN {X 0,Y 438.209,Z 480.447,A -85,B 0,C 180,E1 -18383.25,E2 -18383.25} C_VEL
LIN {X 0,Y 444.561,Z 490.845,A -85,B 0,C 180,E1 -18385.549,E2 -18385.549} C_VEL
LIN {X 0,Y 452.035,Z 503.617,A -85,B 0,C 180,E1 -18387.966,E2 -18387.966} C_VEL
LIN {X 0,Y 459.559,Z 517.473,A -85,B 0,C 180,E1 -18390.172,E2 -18390.172} C_VEL
LIN {X 0,Y 460.135,Z 518.947,A -85,B 0,C 180,E1 -18390.345,E2 -18390.345} C_VEL
LIN {X 0,Y 444.218,Z 756.125,A -85,B 0,C 180,E1 -18394.169,E2 -18394.169} C_VEL
LIN {X 0,Y 441.424,Z 781.083,A -85,B 0,C 180,E1 -18394.682,E2 -18394.682} C_VEL
LIN {X 0,Y 437.519,Z 804.565,A -85,B 0,C 180,E1 -18395.333,E2 -18395.333} C_VEL
LIN {X 0,Y 432.836,Z 827.708,A -85,B 0,C 180,E1 -18396.16,E2 -18396.16} C_VEL
LIN {X 0,Y 427.311,Z 849.938,A -85,B 0,C 180,E1 -18397.179,E2 -18397.179} C_VEL
LIN {X 0,Y 421.976,Z 868.984,A -85,B 0,C 180,E1 -18398.233,E2 -18398.233} C_VEL
LIN {X 0,Y 414.527,Z 892.437,A -85,B 0,C 180,E1 -18399.802,E2 -18399.802} C_VEL
LIN {X 0,Y 407.952,Z 911.044,A -85,B 0,C 180,E1 -18401.303,E2 -18401.303} C_VEL
LIN {X 0,Y 400.174,Z 931.449,A -85,B 0,C 180,E1 -18403.251,E2 -18403.251} C_VEL
LIN {X 0,Y 393.017,Z 948.732,A -85,B 0,C 180,E1 -18405.22,E2 -18405.22} C_VEL
LIN {X 0,Y 385.807,Z 965.442,A -85,B 0,C 180,E1 -18407.435,E2 -18407.435} C_VEL
LIN {X 0,Y 377.909,Z 982.883,A -85,B 0,C 180,E1 -18410.186,E2 -18410.186} C_VEL
LIN {X 0,Y 371.316,Z 997.234,A -85,B 0,C 180,E1 -18412.852,E2 -18412.852} C_VEL
LIN {X 0,Y 364.413,Z 1012.203,A -85,B 0,C 180,E1 -18416.151,E2 -18416.151} C_VEL
LIN {X 0,Y 359.157,Z 1023.818,A -85,B 0,C 180,E1 -18419.186,E2 -18419.186} C_VEL
LIN {X 0,Y 353.965,Z 1035.972,A -85,B 0,C 180,E1 -18422.948,E2 -18422.948} C_VEL
LIN {X 0,Y 350.283,Z 1045.282,A -85,B 0,C 180,E1 -18426.445,E2 -18426.445} C_VEL
LIN {X 0,Y 347.367,Z 1053.9,A -85,B 0,C 180,E1 -18430.319,E2 -18430.319} C_VEL
LIN {X 0,Y 345.47,Z 1060.656,A -85,B 0,C 180,E1 -18434.213,E2 -18434.213} C_VEL
LIN {X 0,Y 344.491,Z 1065.534,A -85,B 0,C 180,E1 -18437.767,E2 -18437.767} C_VEL
LIN {X 0,Y 344.018,Z 1069.54,A -85,B 0,C 180,E1 -18441.812,E2 -18441.812} C_VEL
LIN {X 0,Y 343.956,Z 1071.582,A -85,B 0,C 180,E1 -18445.164,E2 -18445.164} C_VEL
LIN {X 0,Y 343.967,Z 1072.51,A -85,B 0,C 180,E1 -18448.334,E2 -18448.334} C_VEL
LIN {X 0,Y 343.971,Z 1072.443,A -85,B 0,C 180,E1 -18451.499,E2 -18451.499} C_VEL
LIN {X 0,Y 343.962,Z 1071.164,A -85,B 0,C 180,E1 -18455.17,E2 -18455.17} C_VEL
LIN {X 0,Y 344.07,Z 1068.196,A -85,B 0,C 180,E1 -18459.029,E2 -18459.029} C_VEL
LIN {X 0,Y 344.508,Z 1064.445,A -85,B 0,C 180,E1 -18462.402,E2 -18462.402} C_VEL
LIN {X 0,Y 345.679,Z 1058.425,A -85,B 0,C 180,E1 -18466.467,E2 -18466.467} C_VEL
LIN {X 0,Y 347.575,Z 1051.212,A -85,B 0,C 180,E1 -18470.195,E2 -18470.195} C_VEL
LIN {X 0,Y 350.422,Z 1042.532,A -85,B 0,C 180,E1 -18473.902,E2 -18473.902} C_VEL
LIN {X 0,Y 354.414,Z 1031.767,A -85,B 0,C 180,E1 -18477.64,E2 -18477.64} C_VEL
LIN {X 0,Y 358.922,Z 1020.654,A -85,B 0,C 180,E1 -18480.903,E2 -18480.903} C_VEL
LIN {X 0,Y 364.889,Z 1006.574,A -85,B 0,C 180,E1 -18484.367,E2 -18484.367} C_VEL
LIN {X 0,Y 370.7,Z 993.128,A -85,B 0,C 180,E1 -18487.171,E2 -18487.171} C_VEL
LIN {X 0,Y 378.081,Z 976.039,A -85,B 0,C 180,E1 -18490.188,E2 -18490.188} C_VEL
LIN {X 0,Y 384.649,Z 960.401,A -85,B 0,C 180,E1 -18492.521,E2 -18492.521} C_VEL
LIN {X 0,Y 392.269,Z 941.612,A -85,B 0,C 180,E1 -18494.916,E2 -18494.916} C_VEL
LIN {X 0,Y 399.107,Z 923.548,A -85,B 0,C 180,E1 -18496.847,E2 -18496.847} C_VEL
LIN {X 0,Y 406.178,Z 903.709,A -85,B 0,C 180,E1 -18498.661,E2 -18498.661} C_VEL
LIN {X 0,Y 413.066,Z 882.274,A -85,B 0,C 180,E1 -18500.279,E2 -18500.279} C_VEL
LIN {X 0,Y 418.84,Z 862.438,A -85,B 0,C 180,E1 -18501.539,E2 -18501.539} C_VEL
LIN {X 0,Y 424.997,Z 838.146,A -85,B 0,C 180,E1 -18502.797,E2 -18502.797} C_VEL
LIN {X 0,Y 429.429,Z 817.828,A -85,B 0,C 180,E1 -18503.641,E2 -18503.641} C_VEL
LIN {X 0,Y 433.907,Z 792.97,A -85,B 0,C 180,E1 -18504.456,E2 -18504.456} C_VEL
LIN {X 0,Y 436.925,Z 770.642,A -85,B 0,C 180,E1 -18505.005,E2 -18505.005} C_VEL
LIN {X 0,Y 439.222,Z 744.431,A -85,B 0,C 180,E1 -18505.5,E2 -18505.5} C_VEL
LIN {X 0,Y 453.782,Z 514.45,A -85,B 0,C 180,E1 -18509.228,E2 -18509.228} C_VEL
LIN {X 0,Y 445.888,Z 499.814,A -85,B 0,C 180,E1 -18511.358,E2 -18511.358} C_VEL
LIN {X 0,Y 439.016,Z 487.752,A -85,B 0,C 180,E1 -18513.377,E2 -18513.377} C_VEL
LIN {X 0,Y 431.635,Z 475.607,A -85,B 0,C 180,E1 -18515.757,E2 -18515.757} C_VEL
LIN {X 0,Y 424.599,Z 464.616,A -85,B 0,C 180,E1 -18518.302,E2 -18518.302} C_VEL
LIN {X 0,Y 420.526,Z 459.198,A -85,B 0,C 180,E1 -18519.905,E2 -18519.905} C_VEL
LIN {X 0,Y 417.178,Z 454.774,A -85,B 0,C 180,E1 -18521.339,E2 -18521.339} C_VEL
LIN {X 0,Y 413.242,Z 449.64,A -85,B 0,C 180,E1 -18523.193,E2 -18523.193} C_VEL
LIN {X 0,Y 409.203,Z 444.449,A -85,B 0,C 180,E1 -18525.351,E2 -18525.351} C_VEL
LIN {X 0,Y 405.851,Z 440.426,A -85,B 0,C 180,E1 -18527.406,E2 -18527.406} C_VEL
LIN {X 0,Y 404.77,Z 438.815,A -85,B 0,C 180,E1 -18528.169,E2 -18528.169} C_VEL
LIN {X 0,Y 401.587,Z 435.541,A -85,B 0,C 180,E1 -18530.614,E2 -18530.614} C_VEL
LIN {X 0,Y 400.27,Z 432.932,A -85,B 0,C 180,E1 -18531.958,E2 -18531.958} C_VEL
LIN {X 0,Y 396.63,Z 429.723,A -85,B 0,C 180,E1 -18536.821,E2 -18536.821} C_VEL
LIN {X 0,Y 395.824,Z 426.96,A -85,B 0,C 180,E1 -18540.724,E2 -18540.724} C_VEL
LIN {X 0,Y 395.829,Z 427.125,A -85,B 0,C 180,E1 -18542.027,E2 -18542.027} C_VEL
LIN {X 0,Y 399.586,Z 432.613,A -85,B 0,C 180,E1 -18549.797,E2 -18549.797} C_VEL
LIN {X 0,Y 400.45,Z 433.228,A -85,B 0,C 180,E1 -18550.648,E2 -18550.648} C_VEL
LIN {X 0,Y 402.899,Z 437.235,A -85,B 0,C 180,E1 -18552.906,E2 -18552.906} C_VEL
LIN {X 0,Y 405.348,Z 439.459,A -85,B 0,C 180,E1 -18554.646,E2 -18554.646} C_VEL
LIN {X 0,Y 408.565,Z 443.897,A -85,B 0,C 180,E1 -18556.712,E2 -18556.712} C_VEL
LIN {X 0,Y 410.133,Z 445.616,A -85,B 0,C 180,E1 -18557.59,E2 -18557.59} C_VEL
LIN {X 0,Y 413.78,Z 450.151,A -85,B 0,C 180,E1 -18559.48,E2 -18559.48} C_VEL
LIN {X 0,Y 419.127,Z 457.248,A -85,B 0,C 180,E1 -18561.923,E2 -18561.923} C_VEL
LIN {X 0,Y 423.598,Z 463.234,A -85,B 0,C 180,E1 -18563.732,E2 -18563.732} C_VEL
LIN {X 0,Y 429.495,Z 471.271,A -85,B 0,C 180,E1 -18565.882,E2 -18565.882} C_VEL
LIN {X 0,Y 438.817,Z 484.724,A -85,B 0,C 180,E1 -18568.886,E2 -18568.886} C_VEL
LIN {X 0,Y 447.84,Z 498.76,A -85,B 0,C 180,E1 -18571.46,E2 -18571.46} C_VEL
LIN {X 0,Y 454.002,Z 508.927,A -85,B 0,C 180,E1 -18573.072,E2 -18573.072} C_VEL
LIN {X 0,Y 438.923,Z 743.104,A -85,B 0,C 180,E1 -18576.874,E2 -18576.874} C_VEL
LIN {X 0,Y 436.313,Z 767.847,A -85,B 0,C 180,E1 -18577.41,E2 -18577.41} C_VEL
LIN {X 0,Y 432.881,Z 790.351,A -85,B 0,C 180,E1 -18578.081,E2 -18578.081} C_VEL
LIN {X 0,Y 428.949,Z 811.404,A -85,B 0,C 180,E1 -18578.871,E2 -18578.871} C_VEL
LIN {X 0,Y 423.547,Z 835.184,A -85,B 0,C 180,E1 -18579.998,E2 -18579.998} C_VEL
LIN {X 0,Y 418.294,Z 855.147,A -85,B 0,C 180,E1 -18581.151,E2 -18581.151} C_VEL
LIN {X 0,Y 411.333,Z 878.308,A -85,B 0,C 180,E1 -18582.767,E2 -18582.767} C_VEL
LIN {X 0,Y 405.192,Z 896.671,A -85,B 0,C 180,E1 -18584.305,E2 -18584.305} C_VEL
LIN {X 0,Y 397.655,Z 917.383,A -85,B 0,C 180,E1 -18586.353,E2 -18586.353} C_VEL
LIN {X 0,Y 390.791,Z 934.743,A -85,B 0,C 180,E1 -18588.397,E2 -18588.397} C_VEL
LIN {X 0,Y 383.383,Z 952.654,A -85,B 0,C 180,E1 -18590.865,E2 -18590.865} C_VEL
LIN {X 0,Y 376.393,Z 968.563,A -85,B 0,C 180,E1 -18593.483,E2 -18593.483} C_VEL
LIN {X 0,Y 369.506,Z 984.177,A -85,B 0,C 180,E1 -18596.494,E2 -18596.494} C_VEL
LIN {X 0,Y 363.474,Z 997.527,A -85,B 0,C 180,E1 -18599.591,E2 -18599.591} C_VEL
LIN {X 0,Y 358.039,Z 1010.001,A -85,B 0,C 180,E1 -18602.983,E2 -18602.983} C_VEL
LIN {X 0,Y 353.35,Z 1021.095,A -85,B 0,C 180,E1 -18606.661,E2 -18606.661} C_VEL
LIN {X 0,Y 349.871,Z 1030.252,A -85,B 0,C 180,E1 -18610.292,E2 -18610.292} C_VEL
LIN {X 0,Y 347.139,Z 1038.31,A -85,B 0,C 180,E1 -18614.291,E2 -18614.291} C_VEL
LIN {X 0,Y 345.575,Z 1043.981,A -85,B 0,C 180,E1 -18617.806,E2 -18617.806} C_VEL
LIN {X 0,Y 344.518,Z 1049.06,A -85,B 0,C 180,E1 -18621.992,E2 -18621.992} C_VEL
LIN {X 0,Y 344.132,Z 1051.951,A -85,B 0,C 180,E1 -18625.501,E2 -18625.501} C_VEL
LIN {X 0,Y 344.007,Z 1053.643,A -85,B 0,C 180,E1 -18628.834,E2 -18628.834} C_VEL
LIN {X 0,Y 343.975,Z 1054.3,A -85,B 0,C 180,E1 -18632.666,E2 -18632.666} C_VEL
LIN {X 0,Y 344.048,Z 1053.512,A -85,B 0,C 180,E1 -18636.341,E2 -18636.341} C_VEL
LIN {X 0,Y 344.246,Z 1051.729,A -85,B 0,C 180,E1 -18639.699,E2 -18639.699} C_VEL
LIN {X 0,Y 344.911,Z 1048.144,A -85,B 0,C 180,E1 -18643.793,E2 -18643.793} C_VEL
LIN {X 0,Y 346.175,Z 1043.221,A -85,B 0,C 180,E1 -18647.603,E2 -18647.603} C_VEL
LIN {X 0,Y 348.252,Z 1036.964,A -85,B 0,C 180,E1 -18651.385,E2 -18651.385} C_VEL
LIN {X 0,Y 351.392,Z 1028.741,A -85,B 0,C 180,E1 -18655.266,E2 -18655.266} C_VEL
LIN {X 0,Y 355.068,Z 1020.179,A -85,B 0,C 180,E1 -18658.602,E2 -18658.602} C_VEL
LIN {X 0,Y 360.682,Z 1007.932,A -85,B 0,C 180,E1 -18662.535,E2 -18662.535} C_VEL
LIN {X 0,Y 366.074,Z 996.554,A -85,B 0,C 180,E1 -18665.576,E2 -18665.576} C_VEL
LIN {X 0,Y 373.395,Z 981.283,A -85,B 0,C 180,E1 -18668.998,E2 -18668.998} C_VEL
LIN {X 0,Y 379.819,Z 967.675,A -85,B 0,C 180,E1 -18671.56,E2 -18671.56} C_VEL
LIN {X 0,Y 387.778,Z 950.382,A -85,B 0,C 180,E1 -18674.329,E2 -18674.329} C_VEL
LIN {X 0,Y 388.217,Z 949.36,A -85,B 0,C 180,E1 -18674.474,E2 -18674.474} C_VEL
LIN {X 0,Y 389.76,Z 944.239,A -85,B 0,C 180,E1 -18675.303,E2 -18675.303} C_VEL
LIN {X 0,Y 391.097,Z 931.691,A -85,B 0,C 180,E1 -18677.605,E2 -18677.605} C_VEL
LIN {X 0,Y 392.745,Z 926.172,A -85,B 0,C 180,E1 -18678.363,E2 -18678.363} C_VEL
LIN {X 0,Y 399.955,Z 908.591,A -85,B 0,C 180,E1 -18680.242,E2 -18680.242} C_VEL
LIN {X 0,Y 407.507,Z 888.86,A -85,B 0,C 180,E1 -18682.042,E2 -18682.042} C_VEL
LIN {X 0,Y 414.514,Z 868.19,A -85,B 0,C 180,E1 -18683.601,E2 -18683.601} C_VEL
LIN {X 0,Y 420.913,Z 847.335,A -85,B 0,C 180,E1 -18684.922,E2 -18684.922} C_VEL
LIN {X 0,Y 426.843,Z 824.704,A -85,B 0,C 180,E1 -18686.096,E2 -18686.096} C_VEL
LIN {X 0,Y 431.447,Z 804.13,A -85,B 0,C 180,E1 -18686.968,E2 -18686.968} C_VEL
LIN {X 0,Y 436.215,Z 777.819,A -85,B 0,C 180,E1 -18687.836,E2 -18687.836} C_VEL
LIN {X 0,Y 439.209,Z 755.869,A -85,B 0,C 180,E1 -18688.376,E2 -18688.376} C_VEL
LIN {X 0,Y 441.994,Z 723.365,A -85,B 0,C 180,E1 -18688.958,E2 -18688.958} C_VEL
LIN {X 0,Y 456.124,Z 517.378,A -85,B 0,C 180,E1 -18692.271,E2 -18692.271} C_VEL
LIN {X 0,Y 448.66,Z 505.374,A -85,B 0,C 180,E1 -18694.489,E2 -18694.489} C_VEL
LIN {X 0,Y 441.538,Z 494.436,A -85,B 0,C 180,E1 -18696.84,E2 -18696.84} C_VEL
LIN {X 0,Y 434.272,Z 483.973,A -85,B 0,C 180,E1 -18699.549,E2 -18699.549} C_VEL
LIN {X 0,Y 428.586,Z 475.918,A -85,B 0,C 180,E1 -18701.994,E2 -18701.994} C_VEL
LIN {X 0,Y 424.21,Z 470.199,A -85,B 0,C 180,E1 -18704.132,E2 -18704.132} C_VEL
LIN {X 0,Y 420.706,Z 465.425,A -85,B 0,C 180,E1 -18706.111,E2 -18706.111} C_VEL
LIN {X 0,Y 417.351,Z 460.927,A -85,B 0,C 180,E1 -18708.32,E2 -18708.32} C_VEL
LIN {X 0,Y 413.336,Z 455.914,A -85,B 0,C 180,E1 -18711.654,E2 -18711.654} C_VEL
LIN {X 0,Y 412.586,Z 454.544,A -85,B 0,C 180,E1 -18712.48,E2 -18712.48} C_VEL
LIN {X 0,Y 408.866,Z 449.156,A -85,B 0,C 180,E1 -18720.56,E2 -18720.56} C_VEL
LIN {X 0,Y 408.943,Z 449.941,A -85,B 0,C 180,E1 -18722.522,E2 -18722.522} C_VEL
LIN {X 0,Y 412.932,Z 454.919,A -85,B 0,C 180,E1 -18729.548,E2 -18729.548} C_VEL
LIN {X 0,Y 415.285,Z 458.851,A -85,B 0,C 180,E1 -18731.809,E2 -18731.809} C_VEL
LIN {X 0,Y 417.379,Z 460.963,A -85,B 0,C 180,E1 -18733.367,E2 -18733.367} C_VEL
LIN {X 0,Y 420.627,Z 465.387,A -85,B 0,C 180,E1 -18735.511,E2 -18735.511} C_VEL
LIN {X 0,Y 421.981,Z 467.163,A -85,B 0,C 180,E1 -18736.307,E2 -18736.307} C_VEL
LIN {X 0,Y 425.927,Z 472.402,A -85,B 0,C 180,E1 -18738.406,E2 -18738.406} C_VEL
LIN {X 0,Y 430.119,Z 478.213,A -85,B 0,C 180,E1 -18740.373,E2 -18740.373} C_VEL
LIN {X 0,Y 436.387,Z 488.165,A -85,B 0,C 180,E1 -18742.996,E2 -18742.996} C_VEL
LIN {X 0,Y 442.221,Z 497.87,A -85,B 0,C 180,E1 -18745.156,E2 -18745.156} C_VEL
LIN {X 0,Y 449.466,Z 510.541,A -85,B 0,C 180,E1 -18747.563,E2 -18747.563} C_VEL
LIN {X 0,Y 455.955,Z 522.77,A -85,B 0,C 180,E1 -18749.529,E2 -18749.529} C_VEL
LIN {X 0,Y 439.817,Z 756.489,A -85,B 0,C 180,E1 -18753.304,E2 -18753.304} C_VEL
LIN {X 0,Y 436.861,Z 781.805,A -85,B 0,C 180,E1 -18753.83,E2 -18753.83} C_VEL
LIN {X 0,Y 432.958,Z 804.698,A -85,B 0,C 180,E1 -18754.465,E2 -18754.465} C_VEL
LIN {X 0,Y 428.149,Z 827.855,A -85,B 0,C 180,E1 -18755.292,E2 -18755.292} C_VEL
LIN {X 0,Y 422.493,Z 850.019,A -85,B 0,C 180,E1 -18756.308,E2 -18756.308} C_VEL
LIN {X 0,Y 416.727,Z 870.035,A -85,B 0,C 180,E1 -18757.42,E2 -18757.42} C_VEL
LIN {X 0,Y 409.383,Z 892.432,A -85,B 0,C 180,E1 -18758.93,E2 -18758.93} C_VEL
LIN {X 0,Y 402.868,Z 910.361,A -85,B 0,C 180,E1 -18760.375,E2 -18760.375} C_VEL
LIN {X 0,Y 394.882,Z 930.781,A -85,B 0,C 180,E1 -18762.321,E2 -18762.321} C_VEL
LIN {X 0,Y 387.308,Z 948.509,A -85,B 0,C 180,E1 -18764.347,E2 -18764.347} C_VEL
LIN {X 0,Y 379.739,Z 965.481,A -85,B 0,C 180,E1 -18766.614,E2 -18766.614} C_VEL
LIN {X 0,Y 371.612,Z 982.773,A -85,B 0,C 180,E1 -18769.372,E2 -18769.372} C_VEL
LIN {X 0,Y 364.666,Z 997.309,A -85,B 0,C 180,E1 -18772.107,E2 -18772.107} C_VEL
LIN {X 0,Y 357.566,Z 1012.065,A -85,B 0,C 180,E1 -18775.412,E2 -18775.412} C_VEL
LIN {X 0,Y 352.066,Z 1023.671,A -85,B 0,C 180,E1 -18778.495,E2 -18778.495} C_VEL
LIN {X 0,Y 346.61,Z 1035.819,A -85,B 0,C 180,E1 -18782.329,E2 -18782.329} C_VEL
LIN {X 0,Y 342.639,Z 1045.323,A -85,B 0,C 180,E1 -18785.98,E2 -18785.98} C_VEL
LIN {X 0,Y 339.517,Z 1054.033,A -85,B 0,C 180,E1 -18790.024,E2 -18790.024} C_VEL
LIN {X 0,Y 337.534,Z 1060.729,A -85,B 0,C 180,E1 -18794.008,E2 -18794.008} C_VEL
LIN {X 0,Y 336.467,Z 1065.837,A -85,B 0,C 180,E1 -18797.879,E2 -18797.879} C_VEL
LIN {X 0,Y 336.008,Z 1069.573,A -85,B 0,C 180,E1 -18801.96,E2 -18801.96} C_VEL
LIN {X 0,Y 335.957,Z 1071.446,A -85,B 0,C 180,E1 -18805.22,E2 -18805.22} C_VEL
LIN {X 0,Y 335.971,Z 1072.323,A -85,B 0,C 180,E1 -18808.465,E2 -18808.465} C_VEL
LIN {X 0,Y 335.972,Z 1072.18,A -85,B 0,C 180,E1 -18811.876,E2 -18811.876} C_VEL
LIN {X 0,Y 335.967,Z 1070.597,A -85,B 0,C 180,E1 -18815.808,E2 -18815.808} C_VEL
LIN {X 0,Y 336.099,Z 1067.797,A -85,B 0,C 180,E1 -18819.417,E2 -18819.417} C_VEL
LIN {X 0,Y 336.6,Z 1063.99,A -85,B 0,C 180,E1 -18822.873,E2 -18822.873} C_VEL
LIN {X 0,Y 337.969,Z 1057.548,A -85,B 0,C 180,E1 -18827.209,E2 -18827.209} C_VEL
LIN {X 0,Y 339.968,Z 1050.585,A -85,B 0,C 180,E1 -18830.847,E2 -18830.847} C_VEL
LIN {X 0,Y 343.204,Z 1041.391,A -85,B 0,C 180,E1 -18834.805,E2 -18834.805} C_VEL
LIN {X 0,Y 347.415,Z 1030.66,A -85,B 0,C 180,E1 -18838.539,E2 -18838.539} C_VEL
LIN {X 0,Y 352.797,Z 1018.196,A -85,B 0,C 180,E1 -18842.197,E2 -18842.197} C_VEL
LIN {X 0,Y 358.69,Z 1004.836,A -85,B 0,C 180,E1 -18845.438,E2 -18845.438} C_VEL
LIN {X 0,Y 365.412,Z 990.063,A -85,B 0,C 180,E1 -18848.501,E2 -18848.501} C_VEL
LIN {X 0,Y 372.605,Z 973.818,A -85,B 0,C 180,E1 -18851.311,E2 -18851.311} C_VEL
LIN {X 0,Y 379.486,Z 957.992,A -85,B 0,C 180,E1 -18853.656,E2 -18853.656} C_VEL
LIN {X 0,Y 387.669,Z 938.151,A -85,B 0,C 180,E1 -18856.129,E2 -18856.129} C_VEL
LIN {X 0,Y 394.697,Z 920.073,A -85,B 0,C 180,E1 -18858.026,E2 -18858.026} C_VEL
LIN {X 0,Y 402.681,Z 897.708,A -85,B 0,C 180,E1 -18859.988,E2 -18859.988} C_VEL
LIN {X 0,Y 408.89,Z 878.636,A -85,B 0,C 180,E1 -18861.379,E2 -18861.379} C_VEL
LIN {X 0,Y 415.881,Z 854.367,A -85,B 0,C 180,E1 -18862.846,E2 -18862.846} C_VEL
LIN {X 0,Y 421.017,Z 833.822,A -85,B 0,C 180,E1 -18863.85,E2 -18863.85} C_VEL
LIN {X 0,Y 426.28,Z 809.101,A -85,B 0,C 180,E1 -18864.817,E2 -18864.817} C_VEL
LIN {X 0,Y 430.085,Z 786.648,A -85,B 0,C 180,E1 -18865.484,E2 -18865.484} C_VEL
LIN {X 0,Y 433.247,Z 761.58,A -85,B 0,C 180,E1 -18866.053,E2 -18866.053} C_VEL
LIN {X 0,Y 437.351,Z 701.198,A -85,B 0,C 180,E1 -18867.066,E2 -18867.066} C_VEL
LIN {X 0,Y 449.348,Z 518.371,A -85,B 0,C 180,E1 -18870.029,E2 -18870.029} C_VEL
LIN {X 0,Y 440.643,Z 502.043,A -85,B 0,C 180,E1 -18872.498,E2 -18872.498} C_VEL
LIN {X 0,Y 431.8,Z 486.707,A -85,B 0,C 180,E1 -18875.293,E2 -18875.293} C_VEL
LIN {X 0,Y 423.506,Z 473.345,A -85,B 0,C 180,E1 -18878.279,E2 -18878.279} C_VEL
LIN {X 0,Y 418.754,Z 466.746,A -85,B 0,C 180,E1 -18880.18,E2 -18880.18} C_VEL
LIN {X 0,Y 415.164,Z 461.972,A -85,B 0,C 180,E1 -18881.754,E2 -18881.754} C_VEL
LIN {X 0,Y 411.589,Z 457.185,A -85,B 0,C 180,E1 -18883.487,E2 -18883.487} C_VEL
LIN {X 0,Y 407.746,Z 452.143,A -85,B 0,C 180,E1 -18885.587,E2 -18885.587} C_VEL
LIN {X 0,Y 404.358,Z 447.962,A -85,B 0,C 180,E1 -18887.722,E2 -18887.722} C_VEL
LIN {X 0,Y 403.394,Z 446.548,A -85,B 0,C 180,E1 -18888.418,E2 -18888.418} C_VEL
LIN {X 0,Y 400.293,Z 443.224,A -85,B 0,C 180,E1 -18890.873,E2 -18890.873} C_VEL
LIN {X 0,Y 399.001,Z 440.764,A -85,B 0,C 180,E1 -18892.223,E2 -18892.223} C_VEL
LIN {X 0,Y 395.27,Z 436.942,A -85,B 0,C 180,E1 -18897.825,E2 -18897.825} C_VEL
LIN {X 0,Y 394.845,Z 434.875,A -85,B 0,C 180,E1 -18900.871,E2 -18900.871} C_VEL
LIN {X 0,Y 394.857,Z 435.17,A -85,B 0,C 180,E1 -18902.177,E2 -18902.177} C_VEL
LIN {X 0,Y 398.484,Z 440.502,A -85,B 0,C 180,E1 -18909.679,E2 -18909.679} C_VEL
LIN {X 0,Y 399.32,Z 441.244,A -85,B 0,C 180,E1 -18910.532,E2 -18910.532} C_VEL
LIN {X 0,Y 401.931,Z 445.323,A -85,B 0,C 180,E1 -18912.938,E2 -18912.938} C_VEL
LIN {X 0,Y 403.969,Z 447.193,A -85,B 0,C 180,E1 -18914.404,E2 -18914.404} C_VEL
LIN {X 0,Y 407.247,Z 451.707,A -85,B 0,C 180,E1 -18916.547,E2 -18916.547} C_VEL
LIN {X 0,Y 408.559,Z 453.198,A -85,B 0,C 180,E1 -18917.299,E2 -18917.299} C_VEL
LIN {X 0,Y 413.123,Z 459.198,A -85,B 0,C 180,E1 -18919.695,E2 -18919.695} C_VEL
LIN {X 0,Y 417.384,Z 464.843,A -85,B 0,C 180,E1 -18921.649,E2 -18921.649} C_VEL
LIN {X 0,Y 421.791,Z 470.84,A -85,B 0,C 180,E1 -18923.469,E2 -18923.469} C_VEL
LIN {X 0,Y 427.518,Z 478.842,A -85,B 0,C 180,E1 -18925.601,E2 -18925.601} C_VEL
LIN {X 0,Y 436.232,Z 491.621,A -85,B 0,C 180,E1 -18928.474,E2 -18928.474} C_VEL
LIN {X 0,Y 445.114,Z 505.677,A -85,B 0,C 180,E1 -18931.071,E2 -18931.071} C_VEL
LIN {X 0,Y 449.528,Z 513.335,A -85,B 0,C 180,E1 -18932.274,E2 -18932.274} C_VEL
LIN {X 0,Y 434.242,Z 743.941,A -85,B 0,C 180,E1 -18936.029,E2 -18936.029} C_VEL
LIN {X 0,Y 431.442,Z 769.257,A -85,B 0,C 180,E1 -18936.586,E2 -18936.586} C_VEL
LIN {X 0,Y 428.047,Z 790.905,A -85,B 0,C 180,E1 -18937.235,E2 -18937.235} C_VEL
LIN {X 0,Y 423.703,Z 813.538,A -85,B 0,C 180,E1 -18938.092,E2 -18938.092} C_VEL
LIN {X 0,Y 418.451,Z 835.747,A -85,B 0,C 180,E1 -18939.159,E2 -18939.159} C_VEL
LIN {X 0,Y 413.066,Z 855.673,A -85,B 0,C 180,E1 -18940.314,E2 -18940.314} C_VEL
LIN {X 0,Y 405.918,Z 878.775,A -85,B 0,C 180,E1 -18941.934,E2 -18941.934} C_VEL
LIN {X 0,Y 399.591,Z 897.159,A -85,B 0,C 180,E1 -18943.483,E2 -18943.483} C_VEL
LIN {X 0,Y 391.848,Z 917.789,A -85,B 0,C 180,E1 -18945.537,E2 -18945.537} C_VEL
LIN {X 0,Y 384.794,Z 935.08,A -85,B 0,C 180,E1 -18947.589,E2 -18947.589} C_VEL
LIN {X 0,Y 377.123,Z 953.017,A -85,B 0,C 180,E1 -18950.087,E2 -18950.087} C_VEL
LIN {X 0,Y 369.893,Z 968.914,A -85,B 0,C 180,E1 -18952.734,E2 -18952.734} C_VEL
LIN {X 0,Y 362.722,Z 984.541,A -85,B 0,C 180,E1 -18955.791,E2 -18955.791} C_VEL
LIN {X 0,Y 356.465,Z 997.846,A -85,B 0,C 180,E1 -18958.927,E2 -18958.927} C_VEL
LIN {X 0,Y 350.875,Z 1010.119,A -85,B 0,C 180,E1 -18962.322,E2 -18962.322} C_VEL
LIN {X 0,Y 346.08,Z 1020.937,A -85,B 0,C 180,E1 -18965.96,E2 -18965.96} C_VEL
LIN {X 0,Y 342.51,Z 1029.741,A -85,B 0,C 180,E1 -18969.493,E2 -18969.493} C_VEL
LIN {X 0,Y 339.439,Z 1038.279,A -85,B 0,C 180,E1 -18973.749,E2 -18973.749} C_VEL
LIN {X 0,Y 337.744,Z 1043.99,A -85,B 0,C 180,E1 -18977.345,E2 -18977.345} C_VEL
LIN {X 0,Y 336.591,Z 1049.144,A -85,B 0,C 180,E1 -18981.63,E2 -18981.63} C_VEL
LIN {X 0,Y 336.153,Z 1052.073,A -85,B 0,C 180,E1 -18985.223,E2 -18985.223} C_VEL
LIN {X 0,Y 336.015,Z 1053.801,A -85,B 0,C 180,E1 -18988.636,E2 -18988.636} C_VEL
LIN {X 0,Y 335.977,Z 1054.542,A -85,B 0,C 180,E1 -18992.388,E2 -18992.388} C_VEL
LIN {X 0,Y 336.051,Z 1053.782,A -85,B 0,C 180,E1 -18996.321,E2 -18996.321} C_VEL
LIN {X 0,Y 336.257,Z 1052.037,A -85,B 0,C 180,E1 -18999.758,E2 -18999.758} C_VEL
LIN {X 0,Y 336.905,Z 1048.765,A -85,B 0,C 180,E1 -19003.735,E2 -19003.735} C_VEL
LIN {X 0,Y 338.233,Z 1043.823,A -85,B 0,C 180,E1 -19007.728,E2 -19007.728} C_VEL
LIN {X 0,Y 340.229,Z 1038.029,A -85,B 0,C 180,E1 -19011.372,E2 -19011.372} C_VEL
LIN {X 0,Y 343.756,Z 1029.296,A -85,B 0,C 180,E1 -19015.683,E2 -19015.683} C_VEL
LIN {X 0,Y 347.805,Z 1020.326,A -85,B 0,C 180,E1 -19019.257,E2 -19019.257} C_VEL
LIN {X 0,Y 353.711,Z 1008.06,A -85,B 0,C 180,E1 -19023.258,E2 -19023.258} C_VEL
LIN {X 0,Y 359.355,Z 996.673,A -85,B 0,C 180,E1 -19026.346,E2 -19026.346} C_VEL
LIN {X 0,Y 366.994,Z 981.38,A -85,B 0,C 180,E1 -19029.812,E2 -19029.812} C_VEL
LIN {X 0,Y 373.667,Z 967.759,A -85,B 0,C 180,E1 -19032.402,E2 -19032.402} C_VEL
LIN {X 0,Y 381.915,Z 950.439,A -85,B 0,C 180,E1 -19035.195,E2 -19035.195} C_VEL
LIN {X 0,Y 389.183,Z 934.285,A -85,B 0,C 180,E1 -19037.38,E2 -19037.38} C_VEL
LIN {X 0,Y 392.745,Z 926.172,A -85,B 0,C 180,E1 -19038.363,E2 -19038.363} C_VEL
LIN {X 0,Y 394.432,Z 920.552,A -85,B 0,C 180,E1 -19039.104,E2 -19039.104} C_VEL
LIN {X 0,Y 396.226,Z 906.857,A -85,B 0,C 180,E1 -19041.226,E2 -19041.226} C_VEL
LIN {X 0,Y 397.892,Z 900.897,A -85,B 0,C 180,E1 -19041.9,E2 -19041.9} C_VEL
LIN {X 0,Y 405.199,Z 881.272,A -85,B 0,C 180,E1 -19043.558,E2 -19043.558} C_VEL
LIN {X 0,Y 412.345,Z 860.319,A -85,B 0,C 180,E1 -19045.046,E2 -19045.046} C_VEL
LIN {X 0,Y 418.746,Z 838.389,A -85,B 0,C 180,E1 -19046.321,E2 -19046.321} C_VEL
LIN {X 0,Y 424.093,Z 817.585,A -85,B 0,C 180,E1 -19047.32,E2 -19047.32} C_VEL
LIN {X 0,Y 429.206,Z 793.384,A -85,B 0,C 180,E1 -19048.246,E2 -19048.246} C_VEL
LIN {X 0,Y 432.677,Z 772.93,A -85,B 0,C 180,E1 -19048.86,E2 -19048.86} C_VEL
LIN {X 0,Y 435.925,Z 747.159,A -85,B 0,C 180,E1 -19049.442,E2 -19049.442} C_VEL
LIN {X 0,Y 442.479,Z 655.953,A -85,B 0,C 180,E1 -19050.938,E2 -19050.938} C_VEL
LIN {X 0,Y 452.005,Z 521.752,A -85,B 0,C 180,E1 -19053.096,E2 -19053.096} C_VEL
LIN {X 0,Y 443.659,Z 508.27,A -85,B 0,C 180,E1 -19055.713,E2 -19055.713} C_VEL
LIN {X 0,Y 436.155,Z 496.857,A -85,B 0,C 180,E1 -19058.375,E2 -19058.375} C_VEL
LIN {X 0,Y 429.722,Z 487.543,A -85,B 0,C 180,E1 -19060.988,E2 -19060.988} C_VEL
LIN {X 0,Y 425.663,Z 481.958,A -85,B 0,C 180,E1 -19062.854,E2 -19062.854} C_VEL
LIN {X 0,Y 422.605,Z 477.743,A -85,B 0,C 180,E1 -19064.422,E2 -19064.422} C_VEL
LIN {X 0,Y 419.172,Z 473.003,A -85,B 0,C 180,E1 -19066.411,E2 -19066.411} C_VEL
LIN {X 0,Y 415.354,Z 467.868,A -85,B 0,C 180,E1 -19069.037,E2 -19069.037} C_VEL
LIN {X 0,Y 412.211,Z 463.859,A -85,B 0,C 180,E1 -19071.772,E2 -19071.772} C_VEL
LIN {X 0,Y 411.481,Z 462.432,A -85,B 0,C 180,E1 -19072.6,E2 -19072.6} C_VEL
LIN {X 0,Y 407.888,Z 457.115,A -85,B 0,C 180,E1 -19080.562,E2 -19080.562} C_VEL
LIN {X 0,Y 407.965,Z 457.915,A -85,B 0,C 180,E1 -19082.529,E2 -19082.529} C_VEL
LIN {X 0,Y 411.813,Z 462.908,A -85,B 0,C 180,E1 -19089.433,E2 -19089.433} C_VEL
LIN {X 0,Y 414.315,Z 466.922,A -85,B 0,C 180,E1 -19091.837,E2 -19091.837} C_VEL
LIN {X 0,Y 416.026,Z 468.681,A -85,B 0,C 180,E1 -19093.128,E2 -19093.128} C_VEL
LIN {X 0,Y 419.324,Z 473.192,A -85,B 0,C 180,E1 -19095.348,E2 -19095.348} C_VEL
LIN {X 0,Y 424.169,Z 479.768,A -85,B 0,C 180,E1 -19098.058,E2 -19098.058} C_VEL
LIN {X 0,Y 428.555,Z 485.995,A -85,B 0,C 180,E1 -19100.165,E2 -19100.165} C_VEL
LIN {X 0,Y 435.127,Z 496.806,A -85,B 0,C 180,E1 -19102.959,E2 -19102.959} C_VEL
LIN {X 0,Y 440.33,Z 505.638,A -85,B 0,C 180,E1 -19104.912,E2 -19104.912} C_VEL
LIN {X 0,Y 447.477,Z 518.495,A -85,B 0,C 180,E1 -19107.335,E2 -19107.335} C_VEL
LIN {X 0,Y 451.836,Z 527.059,A -85,B 0,C 180,E1 -19108.706,E2 -19108.706} C_VEL
LIN {X 0,Y 435.51,Z 756.959,A -85,B 0,C 180,E1 -19112.424,E2 -19112.424} C_VEL
LIN {X 0,Y 432.311,Z 783.047,A -85,B 0,C 180,E1 -19112.973,E2 -19112.973} C_VEL
LIN {X 0,Y 428.415,Z 805.263,A -85,B 0,C 180,E1 -19113.593,E2 -19113.593} C_VEL
LIN {X 0,Y 423.227,Z 829.268,A -85,B 0,C 180,E1 -19114.46,E2 -19114.46} C_VEL
LIN {X 0,Y 417.458,Z 851.23,A -85,B 0,C 180,E1 -19115.475,E2 -19115.475} C_VEL
LIN {X 0,Y 410.858,Z 873.405,A -85,B 0,C 180,E1 -19116.727,E2 -19116.727} C_VEL
LIN {X 0,Y 403.449,Z 894.864,A -85,B 0,C 180,E1 -19118.22,E2 -19118.22} C_VEL
LIN {X 0,Y 395.999,Z 914.671,A -85,B 0,C 180,E1 -19119.862,E2 -19119.862} C_VEL
LIN {X 0,Y 387.554,Z 934.989,A -85,B 0,C 180,E1 -19121.899,E2 -19121.899} C_VEL
LIN {X 0,Y 380.124,Z 951.775,A -85,B 0,C 180,E1 -19123.885,E2 -19123.885} C_VEL
LIN {X 0,Y 371.541,Z 970.057,A -85,B 0,C 180,E1 -19126.453,E2 -19126.453} C_VEL
LIN {X 0,Y 364.131,Z 985.213,A -85,B 0,C 180,E1 -19128.983,E2 -19128.983} C_VEL
LIN {X 0,Y 355.957,Z 1001.627,A -85,B 0,C 180,E1 -19132.239,E2 -19132.239} C_VEL
LIN {X 0,Y 349.489,Z 1014.488,A -85,B 0,C 180,E1 -19135.296,E2 -19135.296} C_VEL
LIN {X 0,Y 343.147,Z 1027.478,A -85,B 0,C 180,E1 -19138.952,E2 -19138.952} C_VEL
LIN {X 0,Y 338.22,Z 1037.972,A -85,B 0,C 180,E1 -19142.536,E2 -19142.536} C_VEL
LIN {X 0,Y 334.078,Z 1047.812,A -85,B 0,C 180,E1 -19146.543,E2 -19146.543} C_VEL
LIN {X 0,Y 331.14,Z 1055.704,A -85,B 0,C 180,E1 -19150.601,E2 -19150.601} C_VEL
LIN {X 0,Y 329.346,Z 1061.84,A -85,B 0,C 180,E1 -19154.504,E2 -19154.504} C_VEL
LIN {X 0,Y 328.314,Z 1066.83,A -85,B 0,C 180,E1 -19158.76,E2 -19158.76} C_VEL
LIN {X 0,Y 327.994,Z 1069.723,A -85,B 0,C 180,E1 -19162.291,E2 -19162.291} C_VEL
LIN {X 0,Y 327.957,Z 1071.451,A -85,B 0,C 180,E1 -19165.629,E2 -19165.629} C_VEL
LIN {X 0,Y 327.979,Z 1072.254,A -85,B 0,C 180,E1 -19169.487,E2 -19169.487} C_VEL
LIN {X 0,Y 327.97,Z 1071.561,A -85,B 0,C 180,E1 -19173.321,E2 -19173.321} C_VEL
LIN {X 0,Y 327.971,Z 1069.903,A -85,B 0,C 180,E1 -19176.653,E2 -19176.653} C_VEL
LIN {X 0,Y 328.173,Z 1067.069,A -85,B 0,C 180,E1 -19180.179,E2 -19180.179} C_VEL
LIN {X 0,Y 328.973,Z 1062.17,A -85,B 0,C 180,E1 -19184.432,E2 -19184.432} C_VEL
LIN {X 0,Y 330.479,Z 1056.049,A -85,B 0,C 180,E1 -19188.34,E2 -19188.34} C_VEL
LIN {X 0,Y 333.018,Z 1048.25,A -85,B 0,C 180,E1 -19192.365,E2 -19192.365} C_VEL
LIN {X 0,Y 336.604,Z 1038.771,A -85,B 0,C 180,E1 -19196.27,E2 -19196.27} C_VEL
LIN {X 0,Y 340.884,Z 1028.721,A -85,B 0,C 180,E1 -19199.745,E2 -19199.745} C_VEL
LIN {X 0,Y 346.941,Z 1015.291,A -85,B 0,C 180,E1 -19203.601,E2 -19203.601} C_VEL
LIN {X 0,Y 352.632,Z 1003.098,A -85,B 0,C 180,E1 -19206.545,E2 -19206.545} C_VEL
LIN {X 0,Y 360.291,Z 986.778,A -85,B 0,C 180,E1 -19209.872,E2 -19209.872} C_VEL
LIN {X 0,Y 367.274,Z 971.597,A -85,B 0,C 180,E1 -19212.467,E2 -19212.467} C_VEL
LIN {X 0,Y 375.424,Z 953.377,A -85,B 0,C 180,E1 -19215.109,E2 -19215.109} C_VEL
LIN {X 0,Y 382.766,Z 935.922,A -85,B 0,C 180,E1 -19217.227,E2 -19217.227} C_VEL
LIN {X 0,Y 390.624,Z 916.247,A -85,B 0,C 180,E1 -19219.26,E2 -19219.26} C_VEL
LIN {X 0,Y 398.069,Z 895.555,A -85,B 0,C 180,E1 -19221.025,E2 -19221.025} C_VEL
LIN {X 0,Y 405.041,Z 874.546,A -85,B 0,C 180,E1 -19222.529,E2 -19222.529} C_VEL
LIN {X 0,Y 411.328,Z 852.711,A -85,B 0,C 180,E1 -19223.809,E2 -19223.809} C_VEL
LIN {X 0,Y 416.631,Z 831.84,A -85,B 0,C 180,E1 -19224.815,E2 -19224.815} C_VEL
LIN {X 0,Y 422.047,Z 806.369,A -85,B 0,C 180,E1 -19225.782,E2 -19225.782} C_VEL
LIN {X 0,Y 425.79,Z 784.423,A -85,B 0,C 180,E1 -19226.418,E2 -19226.418} C_VEL
LIN {X 0,Y 429.024,Z 757.571,A -85,B 0,C 180,E1 -19227.002,E2 -19227.002} C_VEL
LIN {X 0,Y 444.359,Z 531.396,A -85,B 0,C 180,E1 -19230.703,E2 -19230.703} C_VEL
LIN {X 0,Y 444.913,Z 522.26,A -85,B 0,C 180,E1 -19230.867,E2 -19230.867} C_VEL
LIN {X 0,Y 436.81,Z 506.792,A -85,B 0,C 180,E1 -19233.269,E2 -19233.269} C_VEL
LIN {X 0,Y 427.783,Z 491.002,A -85,B 0,C 180,E1 -19236.258,E2 -19236.258} C_VEL
LIN {X 0,Y 420.29,Z 478.9,A -85,B 0,C 180,E1 -19239.093,E2 -19239.093} C_VEL
LIN {X 0,Y 414.338,Z 470.487,A -85,B 0,C 180,E1 -19241.644,E2 -19241.644} C_VEL
LIN {X 0,Y 409.552,Z 464.294,A -85,B 0,C 180,E1 -19243.985,E2 -19243.985} C_VEL
LIN {X 0,Y 406.178,Z 459.729,A -85,B 0,C 180,E1 -19245.894,E2 -19245.894} C_VEL
LIN {X 0,Y 402.878,Z 455.499,A -85,B 0,C 180,E1 -19248.04,E2 -19248.04} C_VEL
LIN {X 0,Y 402.026,Z 454.278,A -85,B 0,C 180,E1 -19248.669,E2 -19248.669} C_VEL
LIN {X 0,Y 398.936,Z 450.781,A -85,B 0,C 180,E1 -19251.206,E2 -19251.206} C_VEL
LIN {X 0,Y 397.885,Z 448.657,A -85,B 0,C 180,E1 -19252.346,E2 -19252.346} C_VEL
LIN {X 0,Y 394.206,Z 444.697,A -85,B 0,C 180,E1 -19258.11,E2 -19258.11} C_VEL
LIN {X 0,Y 393.868,Z 442.79,A -85,B 0,C 180,E1 -19261.018,E2 -19261.018} C_VEL
LIN {X 0,Y 393.946,Z 443.622,A -85,B 0,C 180,E1 -19262.958,E2 -19262.958} C_VEL
LIN {X 0,Y 397.248,Z 448.311,A -85,B 0,C 180,E1 -19269.416,E2 -19269.416} C_VEL
LIN {X 0,Y 398.131,Z 449.096,A -85,B 0,C 180,E1 -19270.345,E2 -19270.345} C_VEL
LIN {X 0,Y 400.964,Z 453.399,A -85,B 0,C 180,E1 -19272.97,E2 -19272.97} C_VEL
LIN {X 0,Y 402.689,Z 455.096,A -85,B 0,C 180,E1 -19274.23,E2 -19274.23} C_VEL
LIN {X 0,Y 406.051,Z 459.628,A -85,B 0,C 180,E1 -19276.45,E2 -19276.45} C_VEL
LIN {X 0,Y 407.763,Z 461.997,A -85,B 0,C 180,E1 -19277.459,E2 -19277.459} C_VEL
LIN {X 0,Y 411.333,Z 466.572,A -85,B 0,C 180,E1 -19279.342,E2 -19279.342} C_VEL
LIN {X 0,Y 415.725,Z 472.537,A -85,B 0,C 180,E1 -19281.407,E2 -19281.407} C_VEL
LIN {X 0,Y 421.481,Z 480.366,A -85,B 0,C 180,E1 -19283.785,E2 -19283.785} C_VEL
LIN {X 0,Y 430.54,Z 493.714,A -85,B 0,C 180,E1 -19287.04,E2 -19287.04} C_VEL
LIN {X 0,Y 439.319,Z 507.498,A -85,B 0,C 180,E1 -19289.785,E2 -19289.785} C_VEL
LIN {X 0,Y 445.169,Z 517.392,A -85,B 0,C 180,E1 -19291.454,E2 -19291.454} C_VEL
LIN {X 0,Y 429.649,Z 744.88,A -85,B 0,C 180,E1 -19295.167,E2 -19295.167} C_VEL
LIN {X 0,Y 426.548,Z 771.399,A -85,B 0,C 180,E1 -19295.763,E2 -19295.763} C_VEL
LIN {X 0,Y 423.15,Z 792.357,A -85,B 0,C 180,E1 -19296.401,E2 -19296.401} C_VEL
LIN {X 0,Y 418.528,Z 815.533,A -85,B 0,C 180,E1 -19297.292,E2 -19297.292} C_VEL
LIN {X 0,Y 413.155,Z 837.428,A -85,B 0,C 180,E1 -19298.36,E2 -19298.36} C_VEL
LIN {X 0,Y 407.082,Z 859.179,A -85,B 0,C 180,E1 -19299.643,E2 -19299.643} C_VEL
LIN {X 0,Y 400.317,Z 880.043,A -85,B 0,C 180,E1 -19301.143,E2 -19301.143} C_VEL
LIN {X 0,Y 393.997,Z 897.864,A -85,B 0,C 180,E1 -19302.656,E2 -19302.656} C_VEL
LIN {X 0,Y 385.872,Z 918.795,A -85,B 0,C 180,E1 -19304.765,E2 -19304.765} C_VEL
LIN {X 0,Y 378.903,Z 935.352,A -85,B 0,C 180,E1 -19306.748,E2 -19306.748} C_VEL
LIN {X 0,Y 370.934,Z 953.38,A -85,B 0,C 180,E1 -19309.282,E2 -19309.282} C_VEL
LIN {X 0,Y 363.458,Z 969.265,A -85,B 0,C 180,E1 -19311.958,E2 -19311.958} C_VEL
LIN {X 0,Y 356.382,Z 984.12,A -85,B 0,C 180,E1 -19314.889,E2 -19314.889} C_VEL
LIN {X 0,Y 349.727,Z 997.709,A -85,B 0,C 180,E1 -19318.119,E2 -19318.119} C_VEL
LIN {X 0,Y 343.928,Z 1009.865,A -85,B 0,C 180,E1 -19321.524,E2 -19321.524} C_VEL
LIN {X 0,Y 338.655,Z 1021.228,A -85,B 0,C 180,E1 -19325.398,E2 -19325.398} C_VEL
LIN {X 0,Y 334.898,Z 1030.023,A -85,B 0,C 180,E1 -19329.006,E2 -19329.006} C_VEL
LIN {X 0,Y 331.657,Z 1038.544,A -85,B 0,C 180,E1 -19333.357,E2 -19333.357} C_VEL
LIN {X 0,Y 329.864,Z 1044.246,A -85,B 0,C 180,E1 -19337.038,E2 -19337.038} C_VEL
LIN {X 0,Y 328.633,Z 1049.39,A -85,B 0,C 180,E1 -19341.433,E2 -19341.433} C_VEL
LIN {X 0,Y 328.166,Z 1052.305,A -85,B 0,C 180,E1 -19345.106,E2 -19345.106} C_VEL
LIN {X 0,Y 328.019,Z 1054.025,A -85,B 0,C 180,E1 -19348.603,E2 -19348.603} C_VEL
LIN {X 0,Y 327.98,Z 1054.756,A -85,B 0,C 180,E1 -19352.446,E2 -19352.446} C_VEL
LIN {X 0,Y 328.061,Z 1053.985,A -85,B 0,C 180,E1 -19356.475,E2 -19356.475} C_VEL
LIN {X 0,Y 328.284,Z 1052.234,A -85,B 0,C 180,E1 -19359.998,E2 -19359.998} C_VEL
LIN {X 0,Y 329.029,Z 1048.812,A -85,B 0,C 180,E1 -19364.206,E2 -19364.206} C_VEL
LIN {X 0,Y 330.509,Z 1043.751,A -85,B 0,C 180,E1 -19368.339,E2 -19368.339} C_VEL
LIN {X 0,Y 332.865,Z 1037.506,A -85,B 0,C 180,E1 -19372.301,E2 -19372.301} C_VEL
LIN {X 0,Y 336.502,Z 1029.05,A -85,B 0,C 180,E1 -19376.469,E2 -19376.469} C_VEL
LIN {X 0,Y 340.822,Z 1020.018,A -85,B 0,C 180,E1 -19380.111,E2 -19380.111} C_VEL
LIN {X 0,Y 346.797,Z 1008.189,A -85,B 0,C 180,E1 -19384.01,E2 -19384.01} C_VEL
LIN {X 0,Y 352.877,Z 996.469,A -85,B 0,C 180,E1 -19387.228,E2 -19387.228} C_VEL
LIN {X 0,Y 360.668,Z 981.476,A -85,B 0,C 180,E1 -19390.655,E2 -19390.655} C_VEL
LIN {X 0,Y 367.6,Z 967.844,A -85,B 0,C 180,E1 -19393.271,E2 -19393.271} C_VEL
LIN {X 0,Y 376.145,Z 950.498,A -85,B 0,C 180,E1 -19396.086,E2 -19396.086} C_VEL
LIN {X 0,Y 383.701,Z 934.237,A -85,B 0,C 180,E1 -19398.296,E2 -19398.296} C_VEL
LIN {X 0,Y 392.054,Z 915.275,A -85,B 0,C 180,E1 -19400.488,E2 -19400.488} C_VEL
LIN {X 0,Y 397.892,Z 900.897,A -85,B 0,C 180,E1 -19401.9,E2 -19401.9} C_VEL
LIN {X 0,Y 399.57,Z 894.838,A -85,B 0,C 180,E1 -19402.557,E2 -19402.557} C_VEL
LIN {X 0,Y 401.539,Z 880.043,A -85,B 0,C 180,E1 -19404.488,E2 -19404.488} C_VEL
LIN {X 0,Y 403.175,Z 873.668,A -85,B 0,C 180,E1 -19405.068,E2 -19405.068} C_VEL
LIN {X 0,Y 409.897,Z 853.186,A -85,B 0,C 180,E1 -19406.413,E2 -19406.413} C_VEL
LIN {X 0,Y 416.193,Z 831.541,A -85,B 0,C 180,E1 -19407.605,E2 -19407.605} C_VEL
LIN {X 0,Y 421.864,Z 808.1,A -85,B 0,C 180,E1 -19408.633,E2 -19408.633} C_VEL
LIN {X 0,Y 426.386,Z 785.736,A -85,B 0,C 180,E1 -19409.414,E2 -19409.414} C_VEL
LIN {X 0,Y 430.208,Z 760.734,A -85,B 0,C 180,E1 -19410.07,E2 -19410.07} C_VEL
LIN {X 0,Y 432.598,Z 738.268,A -85,B 0,C 180,E1 -19410.509,E2 -19410.509} C_VEL
LIN {X 0,Y 447.979,Z 526.259,A -85,B 0,C 180,E1 -19413.933,E2 -19413.933} C_VEL
LIN {X 0,Y 439.532,Z 512.486,A -85,B 0,C 180,E1 -19416.717,E2 -19416.717} C_VEL
LIN {X 0,Y 431.504,Z 500.147,A -85,B 0,C 180,E1 -19419.766,E2 -19419.766} C_VEL
LIN {X 0,Y 424.951,Z 490.677,A -85,B 0,C 180,E1 -19422.683,E2 -19422.683} C_VEL
LIN {X 0,Y 420.889,Z 485.14,A -85,B 0,C 180,E1 -19424.781,E2 -19424.781} C_VEL
LIN {X 0,Y 417.649,Z 480.579,A -85,B 0,C 180,E1 -19426.713,E2 -19426.713} C_VEL
LIN {X 0,Y 414.017,Z 475.592,A -85,B 0,C 180,E1 -19429.283,E2 -19429.283} C_VEL
LIN {X 0,Y 410.905,Z 471.414,A -85,B 0,C 180,E1 -19432.098,E2 -19432.098} C_VEL
LIN {X 0,Y 410.246,Z 470.248,A -85,B 0,C 180,E1 -19432.859,E2 -19432.859} C_VEL
LIN {X 0,Y 406.911,Z 465.074,A -85,B 0,C 180,E1 -19440.563,E2 -19440.563} C_VEL
LIN {X 0,Y 406.969,Z 465.799,A -85,B 0,C 180,E1 -19442.394,E2 -19442.394} C_VEL
LIN {X 0,Y 410.641,Z 470.746,A -85,B 0,C 180,E1 -19449.248,E2 -19449.248} C_VEL
LIN {X 0,Y 413.009,Z 474.635,A -85,B 0,C 180,E1 -19451.592,E2 -19451.592} C_VEL
LIN {X 0,Y 414.68,Z 476.395,A -85,B 0,C 180,E1 -19452.888,E2 -19452.888} C_VEL
LIN {X 0,Y 418.024,Z 480.996,A -85,B 0,C 180,E1 -19455.184,E2 -19455.184} C_VEL
LIN {X 0,Y 422.672,Z 487.53,A -85,B 0,C 180,E1 -19457.84,E2 -19457.84} C_VEL
LIN {X 0,Y 426.717,Z 493.371,A -85,B 0,C 180,E1 -19459.827,E2 -19459.827} C_VEL
LIN {X 0,Y 433.716,Z 505.116,A -85,B 0,C 180,E1 -19462.859,E2 -19462.859} C_VEL
LIN {X 0,Y 441.286,Z 518.517,A -85,B 0,C 180,E1 -19465.68,E2 -19465.68} C_VEL
LIN {X 0,Y 447.828,Z 531.14,A -85,B 0,C 180,E1 -19467.864,E2 -19467.864} C_VEL
LIN {X 0,Y 431.317,Z 757.329,A -85,B 0,C 180,E1 -19471.524,E2 -19471.524} C_VEL
LIN {X 0,Y 427.838,Z 784.421,A -85,B 0,C 180,E1 -19472.1,E2 -19472.1} C_VEL
LIN {X 0,Y 423.888,Z 806.262,A -85,B 0,C 180,E1 -19472.714,E2 -19472.714} C_VEL
LIN {X 0,Y 418.06,Z 831.955,A -85,B 0,C 180,E1 -19473.662,E2 -19473.662} C_VEL
LIN {X 0,Y 412.513,Z 852.441,A -85,B 0,C 180,E1 -19474.622,E2 -19474.622} C_VEL
LIN {X 0,Y 405.328,Z 875.569,A -85,B 0,C 180,E1 -19475.953,E2 -19475.953} C_VEL
LIN {X 0,Y 398.484,Z 894.862,A -85,B 0,C 180,E1 -19477.304,E2 -19477.304} C_VEL
LIN {X 0,Y 390.831,Z 914.648,A -85,B 0,C 180,E1 -19478.945,E2 -19478.945} C_VEL
LIN {X 0,Y 382.147,Z 934.931,A -85,B 0,C 180,E1 -19480.987,E2 -19480.987} C_VEL
LIN {X 0,Y 374.49,Z 951.703,A -85,B 0,C 180,E1 -19482.981,E2 -19482.981} C_VEL
LIN {X 0,Y 365.624,Z 969.96,A -85,B 0,C 180,E1 -19485.565,E2 -19485.565} C_VEL
LIN {X 0,Y 357.949,Z 985.105,A -85,B 0,C 180,E1 -19488.116,E2 -19488.116} C_VEL
LIN {X 0,Y 349.451,Z 1001.499,A -85,B 0,C 180,E1 -19491.408,E2 -19491.408} C_VEL
LIN {X 0,Y 342.714,Z 1014.35,A -85,B 0,C 180,E1 -19494.508,E2 -19494.508} C_VEL
LIN {X 0,Y 336.074,Z 1027.324,A -85,B 0,C 180,E1 -19498.223,E2 -19498.223} C_VEL
LIN {X 0,Y 330.792,Z 1038.04,A -85,B 0,C 180,E1 -19501.962,E2 -19501.962} C_VEL
LIN {X 0,Y 326.517,Z 1047.639,A -85,B 0,C 180,E1 -19505.966,E2 -19505.966} C_VEL
LIN {X 0,Y 323.393,Z 1055.523,A -85,B 0,C 180,E1 -19510.117,E2 -19510.117} C_VEL
LIN {X 0,Y 321.47,Z 1061.654,A -85,B 0,C 180,E1 -19514.115,E2 -19514.115} C_VEL
LIN {X 0,Y 320.346,Z 1066.696,A -85,B 0,C 180,E1 -19518.547,E2 -19518.547} C_VEL
LIN {X 0,Y 319.995,Z 1069.639,A -85,B 0,C 180,E1 -19522.278,E2 -19522.278} C_VEL
LIN {X 0,Y 319.957,Z 1071.386,A -85,B 0,C 180,E1 -19525.878,E2 -19525.878} C_VEL
LIN {X 0,Y 319.988,Z 1072.022,A -85,B 0,C 180,E1 -19529.821,E2 -19529.821} C_VEL
LIN {X 0,Y 319.968,Z 1071.269,A -85,B 0,C 180,E1 -19533.583,E2 -19533.583} C_VEL
LIN {X 0,Y 319.984,Z 1069.557,A -85,B 0,C 180,E1 -19537,E2 -19537} C_VEL
LIN {X 0,Y 320.217,Z 1066.668,A -85,B 0,C 180,E1 -19540.616,E2 -19540.616} C_VEL
LIN {X 0,Y 321.182,Z 1061.399,A -85,B 0,C 180,E1 -19545.159,E2 -19545.159} C_VEL
LIN {X 0,Y 322.786,Z 1055.481,A -85,B 0,C 180,E1 -19548.981,E2 -19548.981} C_VEL
LIN {X 0,Y 325.582,Z 1047.504,A -85,B 0,C 180,E1 -19553.147,E2 -19553.147} C_VEL
LIN {X 0,Y 329.389,Z 1038.022,A -85,B 0,C 180,E1 -19557.087,E2 -19557.087} C_VEL
LIN {X 0,Y 334.287,Z 1027.212,A -85,B 0,C 180,E1 -19560.856,E2 -19560.856} C_VEL
LIN {X 0,Y 340.353,Z 1014.354,A -85,B 0,C 180,E1 -19564.541,E2 -19564.541} C_VEL
LIN {X 0,Y 346.711,Z 1001.36,A -85,B 0,C 180,E1 -19567.69,E2 -19567.69} C_VEL
LIN {X 0,Y 354.366,Z 985.586,A -85,B 0,C 180,E1 -19570.891,E2 -19570.891} C_VEL
LIN {X 0,Y 361.656,Z 970.313,A -85,B 0,C 180,E1 -19573.505,E2 -19573.505} C_VEL
LIN {X 0,Y 370.629,Z 950.761,A -85,B 0,C 180,E1 -19576.304,E2 -19576.304} C_VEL
LIN {X 0,Y 377.757,Z 934.31,A -85,B 0,C 180,E1 -19578.282,E2 -19578.282} C_VEL
LIN {X 0,Y 386.147,Z 913.615,A -85,B 0,C 180,E1 -19580.385,E2 -19580.385} C_VEL
LIN {X 0,Y 392.979,Z 895.121,A -85,B 0,C 180,E1 -19581.951,E2 -19581.951} C_VEL
LIN {X 0,Y 400.135,Z 874.089,A -85,B 0,C 180,E1 -19583.455,E2 -19583.455} C_VEL
LIN {X 0,Y 406.584,Z 852.194,A -85,B 0,C 180,E1 -19584.733,E2 -19584.733} C_VEL
LIN {X 0,Y 411.987,Z 831.39,A -85,B 0,C 180,E1 -19585.732,E2 -19585.732} C_VEL
LIN {X 0,Y 417.472,Z 806.131,A -85,B 0,C 180,E1 -19586.685,E2 -19586.685} C_VEL
LIN {X 0,Y 421.276,Z 784.291,A -85,B 0,C 180,E1 -19587.316,E2 -19587.316} C_VEL
LIN {X 0,Y 424.587,Z 757.418,A -85,B 0,C 180,E1 -19587.9,E2 -19587.9} C_VEL
LIN {X 0,Y 440.342,Z 531.518,A -85,B 0,C 180,E1 -19591.6,E2 -19591.6} C_VEL
LIN {X 0,Y 440.634,Z 526.173,A -85,B 0,C 180,E1 -19591.707,E2 -19591.707} C_VEL
LIN {X 0,Y 432.575,Z 510.753,A -85,B 0,C 180,E1 -19594.206,E2 -19594.206} C_VEL
LIN {X 0,Y 424.816,Z 497.033,A -85,B 0,C 180,E1 -19596.891,E2 -19596.891} C_VEL
LIN {X 0,Y 418.086,Z 485.932,A -85,B 0,C 180,E1 -19599.527,E2 -19599.527} C_VEL
LIN {X 0,Y 412.337,Z 477.708,A -85,B 0,C 180,E1 -19602.063,E2 -19602.063} C_VEL
LIN {X 0,Y 407.928,Z 471.833,A -85,B 0,C 180,E1 -19604.285,E2 -19604.285} C_VEL
LIN {X 0,Y 404.622,Z 467.31,A -85,B 0,C 180,E1 -19606.204,E2 -19606.204} C_VEL
LIN {X 0,Y 401.321,Z 462.864,A -85,B 0,C 180,E1 -19608.43,E2 -19608.43} C_VEL
LIN {X 0,Y 397.458,Z 458.072,A -85,B 0,C 180,E1 -19611.683,E2 -19611.683} C_VEL
LIN {X 0,Y 396.63,Z 456.484,A -85,B 0,C 180,E1 -19612.613,E2 -19612.613} C_VEL
LIN {X 0,Y 393.119,Z 452.323,A -85,B 0,C 180,E1 -19618.543,E2 -19618.543} C_VEL
LIN {X 0,Y 392.894,Z 450.705,A -85,B 0,C 180,E1 -19621.167,E2 -19621.167} C_VEL
LIN {X 0,Y 393.131,Z 452.387,A -85,B 0,C 180,E1 -19623.938,E2 -19623.938} C_VEL
LIN {X 0,Y 396.418,Z 456.356,A -85,B 0,C 180,E1 -19629.583,E2 -19629.583} C_VEL
LIN {X 0,Y 397.008,Z 457.086,A -85,B 0,C 180,E1 -19630.228,E2 -19630.228} C_VEL
LIN {X 0,Y 399.817,Z 461.29,A -85,B 0,C 180,E1 -19632.861,E2 -19632.861} C_VEL
LIN {X 0,Y 401.324,Z 462.818,A -85,B 0,C 180,E1 -19633.985,E2 -19633.985} C_VEL
LIN {X 0,Y 404.74,Z 467.435,A -85,B 0,C 180,E1 -19636.284,E2 -19636.284} C_VEL
LIN {X 0,Y 409.748,Z 474.244,A -85,B 0,C 180,E1 -19639.087,E2 -19639.087} C_VEL
LIN {X 0,Y 413.929,Z 480.014,A -85,B 0,C 180,E1 -19641.096,E2 -19641.096} C_VEL
LIN {X 0,Y 419.585,Z 487.91,A -85,B 0,C 180,E1 -19643.489,E2 -19643.489} C_VEL
LIN {X 0,Y 428.149,Z 500.756,A -85,B 0,C 180,E1 -19646.641,E2 -19646.641} C_VEL
LIN {X 0,Y 436.584,Z 514.241,A -85,B 0,C 180,E1 -19649.348,E2 -19649.348} C_VEL
LIN {X 0,Y 440.881,Z 521.726,A -85,B 0,C 180,E1 -19650.623,E2 -19650.623} C_VEL
LIN {X 0,Y 425.191,Z 745.395,A -85,B 0,C 180,E1 -19654.279,E2 -19654.279} C_VEL
LIN {X 0,Y 421.987,Z 771.99,A -85,B 0,C 180,E1 -19654.879,E2 -19654.879} C_VEL
LIN {X 0,Y 418.53,Z 792.778,A -85,B 0,C 180,E1 -19655.512,E2 -19655.512} C_VEL
LIN {X 0,Y 413.739,Z 816.139,A -85,B 0,C 180,E1 -19656.412,E2 -19656.412} C_VEL
LIN {X 0,Y 408.538,Z 836.869,A -85,B 0,C 180,E1 -19657.419,E2 -19657.419} C_VEL
LIN {X 0,Y 402.594,Z 857.714,A -85,B 0,C 180,E1 -19658.639,E2 -19658.639} C_VEL
LIN {X 0,Y 395.356,Z 879.706,A -85,B 0,C 180,E1 -19660.201,E2 -19660.201} C_VEL
LIN {X 0,Y 388.487,Z 898.569,A -85,B 0,C 180,E1 -19661.807,E2 -19661.807} C_VEL
LIN {X 0,Y 379.969,Z 919.801,A -85,B 0,C 180,E1 -19663.969,E2 -19663.969} C_VEL
LIN {X 0,Y 372.729,Z 936.462,A -85,B 0,C 180,E1 -19665.989,E2 -19665.989} C_VEL
LIN {X 0,Y 364.37,Z 954.654,A -85,B 0,C 180,E1 -19668.598,E2 -19668.598} C_VEL
LIN {X 0,Y 357.091,Z 969.614,A -85,B 0,C 180,E1 -19671.155,E2 -19671.155} C_VEL
LIN {X 0,Y 349.753,Z 984.458,A -85,B 0,C 180,E1 -19674.122,E2 -19674.122} C_VEL
LIN {X 0,Y 342.642,Z 998.396,A -85,B 0,C 180,E1 -19677.496,E2 -19677.496} C_VEL
LIN {X 0,Y 336.519,Z 1010.737,A -85,B 0,C 180,E1 -19681.032,E2 -19681.032} C_VEL
LIN {X 0,Y 331.261,Z 1021.518,A -85,B 0,C 180,E1 -19684.811,E2 -19684.811} C_VEL
LIN {X 0,Y 327.31,Z 1030.305,A -85,B 0,C 180,E1 -19688.495,E2 -19688.495} C_VEL
LIN {X 0,Y 324.001,Z 1038.513,A -85,B 0,C 180,E1 -19692.767,E2 -19692.767} C_VEL
LIN {X 0,Y 322.06,Z 1044.254,A -85,B 0,C 180,E1 -19696.535,E2 -19696.535} C_VEL
LIN {X 0,Y 320.745,Z 1049.314,A -85,B 0,C 180,E1 -19700.852,E2 -19700.852} C_VEL
LIN {X 0,Y 320.194,Z 1052.426,A -85,B 0,C 180,E1 -19704.804,E2 -19704.804} C_VEL
LIN {X 0,Y 320.025,Z 1054.183,A -85,B 0,C 180,E1 -19708.389,E2 -19708.389} C_VEL
LIN {X 0,Y 319.981,Z 1054.932,A -85,B 0,C 180,E1 -19712.149,E2 -19712.149} C_VEL
LIN {X 0,Y 320.057,Z 1054.321,A -85,B 0,C 180,E1 -19716.277,E2 -19716.277} C_VEL
LIN {X 0,Y 320.28,Z 1052.653,A -85,B 0,C 180,E1 -19719.887,E2 -19719.887} C_VEL
LIN {X 0,Y 320.904,Z 1049.772,A -85,B 0,C 180,E1 -19723.698,E2 -19723.698} C_VEL
LIN {X 0,Y 322.467,Z 1044.677,A -85,B 0,C 180,E1 -19728.251,E2 -19728.251} C_VEL
LIN {X 0,Y 324.668,Z 1038.967,A -85,B 0,C 180,E1 -19732.069,E2 -19732.069} C_VEL
LIN {X 0,Y 328.361,Z 1030.807,A -85,B 0,C 180,E1 -19736.397,E2 -19736.397} C_VEL
LIN {X 0,Y 332.715,Z 1021.981,A -85,B 0,C 180,E1 -19740.124,E2 -19740.124} C_VEL
LIN {X 0,Y 338.485,Z 1011.156,A -85,B 0,C 180,E1 -19743.939,E2 -19743.939} C_VEL
LIN {X 0,Y 345.089,Z 998.802,A -85,B 0,C 180,E1 -19747.479,E2 -19747.479} C_VEL
LIN {X 0,Y 352.564,Z 985.141,A -85,B 0,C 180,E1 -19750.779,E2 -19750.779} C_VEL
LIN {X 0,Y 360.305,Z 970.456,A -85,B 0,C 180,E1 -19753.71,E2 -19753.71} C_VEL
LIN {X 0,Y 368.073,Z 955.375,A -85,B 0,C 180,E1 -19756.27,E2 -19756.27} C_VEL
LIN {X 0,Y 376.988,Z 937.051,A -85,B 0,C 180,E1 -19758.873,E2 -19758.873} C_VEL
LIN {X 0,Y 384.682,Z 920.217,A -85,B 0,C 180,E1 -19760.885,E2 -19760.885} C_VEL
LIN {X 0,Y 393.636,Z 898.972,A -85,B 0,C 180,E1 -19763.011,E2 -19763.011} C_VEL
LIN {X 0,Y 400.704,Z 880.424,A -85,B 0,C 180,E1 -19764.56,E2 -19764.56} C_VEL
LIN {X 0,Y 403.175,Z 873.668,A -85,B 0,C 180,E1 -19765.068,E2 -19765.068} C_VEL
LIN {X 0,Y 404.8,Z 867.191,A -85,B 0,C 180,E1 -19765.632,E2 -19765.632} C_VEL
LIN {X 0,Y 406.692,Z 851.349,A -85,B 0,C 180,E1 -19767.363,E2 -19767.363} C_VEL
LIN {X 0,Y 408.136,Z 844.614,A -85,B 0,C 180,E1 -19767.862,E2 -19767.862} C_VEL
LIN {X 0,Y 413.973,Z 823.428,A -85,B 0,C 180,E1 -19768.922,E2 -19768.922} C_VEL
LIN {X 0,Y 419.126,Z 801.682,A -85,B 0,C 180,E1 -19769.814,E2 -19769.814} C_VEL
LIN {X 0,Y 423.683,Z 777.4,A -85,B 0,C 180,E1 -19770.584,E2 -19770.584} C_VEL
LIN {X 0,Y 426.871,Z 755.254,A -85,B 0,C 180,E1 -19771.117,E2 -19771.117} C_VEL
LIN {X 0,Y 429.809,Z 722.524,A -85,B 0,C 180,E1 -19771.694,E2 -19771.694} C_VEL
LIN {X 0,Y 444.069,Z 530.795,A -85,B 0,C 180,E1 -19774.778,E2 -19774.778} C_VEL
LIN {X 0,Y 436.41,Z 518.249,A -85,B 0,C 180,E1 -19777.413,E2 -19777.413} C_VEL
LIN {X 0,Y 429.334,Z 507.17,A -85,B 0,C 180,E1 -19780.201,E2 -19780.201} C_VEL
LIN {X 0,Y 423.024,Z 497.889,A -85,B 0,C 180,E1 -19783.098,E2 -19783.098} C_VEL
LIN {X 0,Y 419.308,Z 492.682,A -85,B 0,C 180,E1 -19785.076,E2 -19785.076} C_VEL
LIN {X 0,Y 416.245,Z 488.267,A -85,B 0,C 180,E1 -19786.95,E2 -19786.95} C_VEL
LIN {X 0,Y 412.688,Z 483.313,A -85,B 0,C 180,E1 -19789.53,E2 -19789.53} C_VEL
LIN {X 0,Y 409.67,Z 479.099,A -85,B 0,C 180,E1 -19792.356,E2 -19792.356} C_VEL
LIN {X 0,Y 409.147,Z 478.135,A -85,B 0,C 180,E1 -19792.981,E2 -19792.981} C_VEL
LIN {X 0,Y 405.936,Z 472.985,A -85,B 0,C 180,E1 -19800.706,E2 -19800.706} C_VEL
LIN {X 0,Y 406.126,Z 474.378,A -85,B 0,C 180,E1 -19803.246,E2 -19803.246} C_VEL
LIN {X 0,Y 409.473,Z 478.582,A -85,B 0,C 180,E1 -19809.062,E2 -19809.062} C_VEL
LIN {X 0,Y 411.873,Z 482.526,A -85,B 0,C 180,E1 -19811.483,E2 -19811.483} C_VEL
LIN {X 0,Y 413.425,Z 484.272,A -85,B 0,C 180,E1 -19812.714,E2 -19812.714} C_VEL
LIN {X 0,Y 417.461,Z 489.989,A -85,B 0,C 180,E1 -19815.49,E2 -19815.49} C_VEL
LIN {X 0,Y 421.183,Z 495.284,A -85,B 0,C 180,E1 -19817.619,E2 -19817.619} C_VEL
LIN {X 0,Y 424.826,Z 500.638,A -85,B 0,C 180,E1 -19819.454,E2 -19819.454} C_VEL
LIN {X 0,Y 432.308,Z 513.406,A -85,B 0,C 180,E1 -19822.758,E2 -19822.758} C_VEL
LIN {X 0,Y 440.672,Z 528.855,A -85,B 0,C 180,E1 -19825.899,E2 -19825.899} C_VEL
LIN {X 0,Y 443.886,Z 535.633,A -85,B 0,C 180,E1 -19827.014,E2 -19827.014} C_VEL
LIN {X 0,Y 427.242,Z 757.597,A -85,B 0,C 180,E1 -19830.605,E2 -19830.605} C_VEL
LIN {X 0,Y 423.71,Z 784.37,A -85,B 0,C 180,E1 -19831.175,E2 -19831.175} C_VEL
LIN {X 0,Y 419.68,Z 806.184,A -85,B 0,C 180,E1 -19831.785,E2 -19831.785} C_VEL
LIN {X 0,Y 413.842,Z 831.412,A -85,B 0,C 180,E1 -19832.708,E2 -19832.708} C_VEL
LIN {X 0,Y 408.322,Z 851.396,A -85,B 0,C 180,E1 -19833.635,E2 -19833.635} C_VEL
LIN {X 0,Y 401.506,Z 873.159,A -85,B 0,C 180,E1 -19834.858,E2 -19834.858} C_VEL
LIN {X 0,Y 393.932,Z 894.049,A -85,B 0,C 180,E1 -19836.304,E2 -19836.304} C_VEL
LIN {X 0,Y 386.349,Z 913.156,A -85,B 0,C 180,E1 -19837.875,E2 -19837.875} C_VEL
LIN {X 0,Y 377.4,Z 933.656,A -85,B 0,C 180,E1 -19839.914,E2 -19839.914} C_VEL
LIN {X 0,Y 369.476,Z 950.519,A -85,B 0,C 180,E1 -19841.908,E2 -19841.908} C_VEL
LIN {X 0,Y 359.799,Z 969.863,A -85,B 0,C 180,E1 -19844.649,E2 -19844.649} C_VEL
LIN {X 0,Y 351.855,Z 984.997,A -85,B 0,C 180,E1 -19847.22,E2 -19847.22} C_VEL
LIN {X 0,Y 342.877,Z 1001.628,A -85,B 0,C 180,E1 -19850.605,E2 -19850.605} C_VEL
LIN {X 0,Y 336.005,Z 1014.213,A -85,B 0,C 180,E1 -19853.688,E2 -19853.688} C_VEL
LIN {X 0,Y 329.057,Z 1027.171,A -85,B 0,C 180,E1 -19857.463,E2 -19857.463} C_VEL
LIN {X 0,Y 323.621,Z 1037.65,A -85,B 0,C 180,E1 -19861.184,E2 -19861.184} C_VEL
LIN {X 0,Y 318.968,Z 1047.503,A -85,B 0,C 180,E1 -19865.379,E2 -19865.379} C_VEL
LIN {X 0,Y 315.623,Z 1055.451,A -85,B 0,C 180,E1 -19869.674,E2 -19869.674} C_VEL
LIN {X 0,Y 313.538,Z 1061.728,A -85,B 0,C 180,E1 -19873.892,E2 -19873.892} C_VEL
LIN {X 0,Y 312.37,Z 1066.613,A -85,B 0,C 180,E1 -19878.38,E2 -19878.38} C_VEL
LIN {X 0,Y 312.001,Z 1069.438,A -85,B 0,C 180,E1 -19882.079,E2 -19882.079} C_VEL
LIN {X 0,Y 311.959,Z 1071.181,A -85,B 0,C 180,E1 -19885.772,E2 -19885.772} C_VEL
LIN {X 0,Y 311.991,Z 1071.805,A -85,B 0,C 180,E1 -19889.816,E2 -19889.816} C_VEL
LIN {X 0,Y 311.968,Z 1071.047,A -85,B 0,C 180,E1 -19893.675,E2 -19893.675} C_VEL
LIN {X 0,Y 311.998,Z 1069.328,A -85,B 0,C 180,E1 -19897.18,E2 -19897.18} C_VEL
LIN {X 0,Y 312.25,Z 1066.432,A -85,B 0,C 180,E1 -19900.89,E2 -19900.89} C_VEL
LIN {X 0,Y 313.297,Z 1061.149,A -85,B 0,C 180,E1 -19905.55,E2 -19905.55} C_VEL
LIN {X 0,Y 315.039,Z 1055.168,A -85,B 0,C 180,E1 -19909.5,E2 -19909.5} C_VEL
LIN {X 0,Y 318.158,Z 1046.817,A -85,B 0,C 180,E1 -19913.917,E2 -19913.917} C_VEL
LIN {X 0,Y 322.247,Z 1037.273,A -85,B 0,C 180,E1 -19917.939,E2 -19917.939} C_VEL
LIN {X 0,Y 327.593,Z 1026.099,A -85,B 0,C 180,E1 -19921.873,E2 -19921.873} C_VEL
LIN {X 0,Y 333.87,Z 1013.402,A -85,B 0,C 180,E1 -19925.521,E2 -19925.521} C_VEL
LIN {X 0,Y 340.927,Z 999.62,A -85,B 0,C 180,E1 -19928.875,E2 -19928.875} C_VEL
LIN {X 0,Y 348.565,Z 984.395,A -85,B 0,C 180,E1 -19931.942,E2 -19931.942} C_VEL
LIN {X 0,Y 356.173,Z 969.031,A -85,B 0,C 180,E1 -19934.574,E2 -19934.574} C_VEL
LIN {X 0,Y 364.98,Z 950.393,A -85,B 0,C 180,E1 -19937.24,E2 -19937.24} C_VEL
LIN {X 0,Y 372.335,Z 933.928,A -85,B 0,C 180,E1 -19939.227,E2 -19939.227} C_VEL
LIN {X 0,Y 381.032,Z 913.033,A -85,B 0,C 180,E1 -19941.351,E2 -19941.351} C_VEL
LIN {X 0,Y 388.104,Z 894.392,A -85,B 0,C 180,E1 -19942.924,E2 -19942.924} C_VEL
LIN {X 0,Y 395.647,Z 872.679,A -85,B 0,C 180,E1 -19944.465,E2 -19944.465} C_VEL
LIN {X 0,Y 402.205,Z 850.772,A -85,B 0,C 180,E1 -19945.725,E2 -19945.725} C_VEL
LIN {X 0,Y 408.035,Z 828.712,A -85,B 0,C 180,E1 -19946.765,E2 -19946.765} C_VEL
LIN {X 0,Y 413.218,Z 804.801,A -85,B 0,C 180,E1 -19947.642,E2 -19947.642} C_VEL
LIN {X 0,Y 417.156,Z 782.419,A -85,B 0,C 180,E1 -19948.278,E2 -19948.278} C_VEL
LIN {X 0,Y 420.314,Z 756.611,A -85,B 0,C 180,E1 -19948.829,E2 -19948.829} C_VEL
LIN {X 0,Y 436.53,Z 530.272,A -85,B 0,C 180,E1 -19952.538,E2 -19952.538} C_VEL
LIN {X 0,Y 428.636,Z 515.087,A -85,B 0,C 180,E1 -19955.099,E2 -19955.099} C_VEL
LIN {X 0,Y 421.73,Z 502.799,A -85,B 0,C 180,E1 -19957.596,E2 -19957.596} C_VEL
LIN {X 0,Y 415.985,Z 493.07,A -85,B 0,C 180,E1 -19959.933,E2 -19959.933} C_VEL
LIN {X 0,Y 410.36,Z 484.919,A -85,B 0,C 180,E1 -19962.487,E2 -19962.487} C_VEL
LIN {X 0,Y 406.316,Z 479.373,A -85,B 0,C 180,E1 -19964.587,E2 -19964.587} C_VEL
LIN {X 0,Y 403.078,Z 474.887,A -85,B 0,C 180,E1 -19966.516,E2 -19966.516} C_VEL
LIN {X 0,Y 399.782,Z 470.229,A -85,B 0,C 180,E1 -19968.823,E2 -19968.823} C_VEL
LIN {X 0,Y 396.394,Z 466.147,A -85,B 0,C 180,E1 -19971.733,E2 -19971.733} C_VEL
LIN {X 0,Y 395.52,Z 464.374,A -85,B 0,C 180,E1 -19972.738,E2 -19972.738} C_VEL
